Yaskawa INFORM job: DEMO_ROOF_SIDE_0625_3PAINT_58.JBI

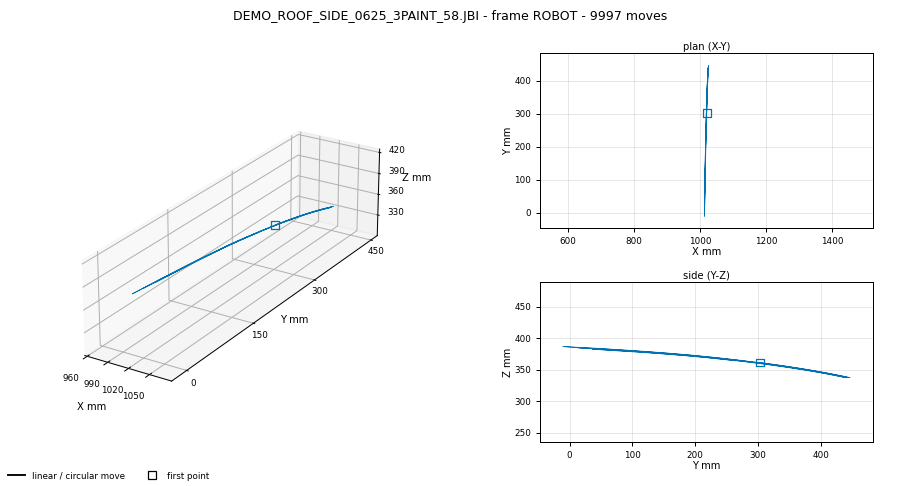
[picture p0: tool path of DEMO_ROOF_SIDE_0625_3PAINT_58.JBI in frame ROBOT, 9997 of 9997 moves have a stored position in this frame; points joined in program order, loops and branches not executed]
/JOB
//NAME DEMO_ROOF_SIDE_0625_3PAINT58
//POS
///NPOS 9997,0,0,0,0,0
///TOOL 0
///USER 0
///POSTYPE ROBOT
///RECTAN
///RCONF 1,0,0,0,0,0,0,0,0,0,0,0,0,0,0,0,0,0,0,0,0,0,0,0
C00000=1019.458,302.892,361.621,170.193,50.128,159.718
C00001=1019.464,303.141,361.589,170.199,50.124,159.718
C00002=1019.471,303.388,361.557,170.204,50.121,159.718
C00003=1019.478,303.636,361.524,170.209,50.117,159.718
C00004=1019.484,303.884,361.492,170.215,50.113,159.718
C00005=1019.491,304.131,361.460,170.220,50.110,159.718
C00006=1019.498,304.379,361.427,170.227,50.106,159.719
C00007=1019.504,304.627,361.396,170.232,50.103,159.719
C00008=1019.511,304.875,361.363,170.237,50.099,159.719
C00009=1019.517,305.122,361.330,170.243,50.095,159.719
C00010=1019.524,305.370,361.299,170.248,50.092,159.719
C00011=1019.530,305.618,361.266,170.255,50.088,159.719
C00012=1019.538,305.866,361.233,170.260,50.085,159.719
C00013=1019.544,306.113,361.201,170.265,50.082,159.719
C00014=1019.550,306.362,361.169,170.271,50.077,159.719
C00015=1019.557,306.609,361.136,170.276,50.074,159.719
C00016=1019.564,306.857,361.103,170.283,50.070,159.720
C00017=1019.570,307.101,361.071,170.288,50.067,159.720
C00018=1019.576,307.344,361.040,170.293,50.064,159.720
C00019=1019.583,307.587,361.008,170.299,50.060,159.720
C00020=1019.590,307.830,360.975,170.305,50.057,159.720
C00021=1019.596,308.074,360.944,170.310,50.053,159.720
C00022=1019.604,308.318,360.911,170.316,50.050,159.720
C00023=1019.610,308.562,360.879,170.322,50.046,159.720
C00024=1019.617,308.805,360.848,170.327,50.043,159.721
C00025=1019.624,309.052,360.815,170.333,50.039,159.721
C00026=1019.630,309.300,360.783,170.338,50.036,159.721
C00027=1019.637,309.548,360.750,170.345,50.033,159.721
C00028=1019.644,309.796,360.717,170.350,50.029,159.721
C00029=1019.650,310.043,360.685,170.356,50.026,159.721
C00030=1019.658,310.291,360.651,170.362,50.023,159.722
C00031=1019.663,310.539,360.618,170.367,50.020,159.722
C00032=1019.669,310.786,360.585,170.373,50.016,159.722
C00033=1019.677,311.034,360.551,170.379,50.013,159.722
C00034=1019.683,311.282,360.518,170.384,50.010,159.722
C00035=1019.689,311.529,360.485,170.391,50.007,159.723
C00036=1019.696,311.777,360.451,170.396,50.004,159.723
C00037=1019.702,312.025,360.418,170.402,50.000,159.723
C00038=1019.709,312.272,360.385,170.408,49.997,159.723
C00039=1019.715,312.520,360.352,170.414,49.994,159.723
C00040=1019.721,312.767,360.318,170.419,49.991,159.724
C00041=1019.728,313.015,360.285,170.425,49.988,159.724
C00042=1019.735,313.263,360.251,170.431,49.984,159.724
C00043=1019.741,313.510,360.218,170.437,49.981,159.724
C00044=1019.748,313.758,360.184,170.443,49.978,159.724
C00045=1019.754,314.006,360.151,170.448,49.976,159.725
C00046=1019.761,314.254,360.117,170.455,49.972,159.725
C00047=1019.768,314.500,360.084,170.460,49.969,159.725
C00048=1019.775,314.749,360.051,170.466,49.967,159.726
C00049=1019.780,314.996,360.017,170.472,49.963,159.726
C00050=1019.788,315.244,359.983,170.478,49.960,159.726
C00051=1019.794,315.491,359.950,170.484,49.957,159.726
C00052=1019.801,315.739,359.916,170.490,49.954,159.727
C00053=1019.807,315.986,359.882,170.495,49.951,159.727
C00054=1019.814,316.235,359.849,170.502,49.948,159.727
C00055=1019.820,316.482,359.816,170.507,49.945,159.727
C00056=1019.828,316.729,359.782,170.514,49.941,159.728
C00057=1019.834,316.977,359.748,170.519,49.939,159.728
C00058=1019.840,317.225,359.715,170.526,49.936,159.728
C00059=1019.848,317.472,359.681,170.532,49.933,159.729
C00060=1019.854,317.719,359.648,170.537,49.930,159.729
C00061=1019.861,317.967,359.613,170.544,49.927,159.729
C00062=1019.868,318.215,359.579,170.549,49.924,159.729
C00063=1019.874,318.462,359.546,170.556,49.921,159.730
C00064=1019.881,318.710,359.513,170.561,49.918,159.730
C00065=1019.888,318.958,359.478,170.568,49.915,159.730
C00066=1019.894,319.205,359.445,170.574,49.912,159.731
C00067=1019.902,319.453,359.411,170.580,49.909,159.731
C00068=1019.909,319.701,359.377,170.586,49.907,159.731
C00069=1019.915,319.949,359.343,170.591,49.903,159.731
C00070=1019.922,320.196,359.309,170.598,49.900,159.732
C00071=1019.929,320.443,359.275,170.603,49.898,159.732
C00072=1019.936,320.691,359.241,170.610,49.895,159.732
C00073=1019.943,320.939,359.207,170.616,49.892,159.733
C00074=1019.950,321.187,359.173,170.622,49.889,159.733
C00075=1019.957,321.434,359.140,170.628,49.886,159.733
C00076=1019.963,321.682,359.106,170.635,49.883,159.734
C00077=1019.971,321.928,359.072,170.640,49.881,159.734
C00078=1019.978,322.174,359.038,170.647,49.878,159.734
C00079=1019.984,322.420,359.004,170.653,49.875,159.735
C00080=1019.991,322.666,358.970,170.659,49.872,159.735
C00081=1019.998,322.912,358.936,170.665,49.869,159.735
C00082=1020.005,323.158,358.902,170.672,49.866,159.736
C00083=1020.012,323.404,358.868,170.677,49.864,159.736
C00084=1020.019,323.650,358.835,170.684,49.861,159.736
C00085=1020.026,323.898,358.800,170.690,49.858,159.737
C00086=1020.033,324.146,358.766,170.696,49.855,159.737
C00087=1020.040,324.393,358.732,170.702,49.853,159.737
C00088=1020.047,324.641,358.697,170.709,49.850,159.738
C00089=1020.054,324.888,358.664,170.715,49.848,159.738
C00090=1020.062,325.135,358.629,170.721,49.845,159.739
C00091=1020.069,325.383,358.595,170.727,49.842,159.739
C00092=1020.075,325.631,358.561,170.734,49.839,159.739
C00093=1020.083,325.878,358.526,170.739,49.836,159.740
C00094=1020.090,326.126,358.492,170.746,49.834,159.740
C00095=1020.097,326.373,358.458,170.753,49.831,159.741
C00096=1020.104,326.621,358.424,170.758,49.828,159.741
C00097=1020.111,326.868,358.388,170.766,49.826,159.741
C00098=1020.118,327.115,358.354,170.771,49.823,159.742
C00099=1020.125,327.363,358.319,170.778,49.821,159.742
C00100=1020.131,327.611,358.284,170.784,49.818,159.743
C00101=1020.139,327.858,358.250,170.791,49.815,159.743
C00102=1020.145,328.106,358.215,170.797,49.813,159.744
C00103=1020.152,328.353,358.180,170.803,49.810,159.744
C00104=1020.159,328.600,358.145,170.809,49.808,159.744
C00105=1020.167,328.848,358.110,170.816,49.806,159.745
C00106=1020.174,329.095,358.075,170.822,49.803,159.745
C00107=1020.181,329.343,358.040,170.829,49.801,159.746
C00108=1020.187,329.591,358.005,170.835,49.798,159.746
C00109=1020.195,329.838,357.971,170.842,49.796,159.747
C00110=1020.201,330.085,357.936,170.848,49.794,159.747
C00111=1020.208,330.333,357.901,170.854,49.791,159.748
C00112=1020.216,330.580,357.866,170.860,49.789,159.748
C00113=1020.223,330.828,357.831,170.867,49.786,159.748
C00114=1020.230,331.075,357.795,170.873,49.784,159.749
C00115=1020.237,331.322,357.760,170.880,49.782,159.750
C00116=1020.244,331.569,357.726,170.887,49.779,159.750
C00117=1020.251,331.818,357.690,170.893,49.777,159.750
C00118=1020.258,332.065,357.655,170.900,49.774,159.751
C00119=1020.265,332.312,357.620,170.906,49.772,159.751
C00120=1020.273,332.560,357.585,170.913,49.770,159.752
C00121=1020.280,332.807,357.550,170.919,49.767,159.752
C00122=1020.287,333.054,357.514,170.925,49.765,159.753
C00123=1020.294,333.301,357.479,170.932,49.763,159.753
C00124=1020.301,333.550,357.443,170.939,49.761,159.754
C00125=1020.308,333.796,357.408,170.946,49.758,159.755
C00126=1020.315,334.044,357.373,170.952,49.756,159.755
C00127=1020.322,334.292,357.337,170.959,49.754,159.756
C00128=1020.329,334.538,357.301,170.965,49.752,159.756
C00129=1020.336,334.786,357.266,170.972,49.750,159.757
C00130=1020.343,335.034,357.231,170.979,49.747,159.757
C00131=1020.351,335.281,357.195,170.985,49.745,159.758
C00132=1020.357,335.528,357.160,170.992,49.743,159.758
C00133=1020.365,335.775,357.123,170.998,49.741,159.759
C00134=1020.372,336.023,357.088,171.005,49.739,159.759
C00135=1020.379,336.270,357.052,171.012,49.736,159.760
C00136=1020.386,336.518,357.017,171.018,49.734,159.760
C00137=1020.393,336.762,356.982,171.025,49.733,159.761
C00138=1020.401,337.005,356.946,171.031,49.731,159.762
C00139=1020.408,337.250,356.911,171.038,49.728,159.762
C00140=1020.415,337.493,356.875,171.044,49.726,159.763
C00141=1020.422,337.737,356.841,171.051,49.724,159.763
C00142=1020.429,337.981,356.806,171.058,49.723,159.764
C00143=1020.436,338.225,356.770,171.065,49.720,159.765
C00144=1020.444,338.469,356.735,171.072,49.718,159.765
C00145=1020.451,338.716,356.699,171.078,49.716,159.766
C00146=1020.459,338.963,356.663,171.085,49.714,159.766
C00147=1020.466,339.211,356.628,171.092,49.712,159.767
C00148=1020.473,339.458,356.592,171.098,49.710,159.768
C00149=1020.480,339.705,356.555,171.106,49.708,159.768
C00150=1020.487,339.953,356.519,171.113,49.706,159.769
C00151=1020.495,340.200,356.483,171.119,49.704,159.770
C00152=1020.502,340.447,356.447,171.126,49.702,159.770
C00153=1020.509,340.695,356.410,171.132,49.701,159.771
C00154=1020.516,340.941,356.374,171.139,49.698,159.771
C00155=1020.524,341.189,356.338,171.147,49.697,159.772
C00156=1020.531,341.436,356.302,171.153,49.695,159.773
C00157=1020.538,341.683,356.265,171.160,49.693,159.773
C00158=1020.545,341.931,356.229,171.167,49.691,159.774
C00159=1020.553,342.178,356.193,171.175,49.689,159.775
C00160=1020.561,342.426,356.157,171.181,49.687,159.775
C00161=1020.567,342.673,356.120,171.188,49.685,159.776
C00162=1020.575,342.919,356.083,171.195,49.684,159.777
C00163=1020.583,343.167,356.047,171.201,49.682,159.777
C00164=1020.590,343.415,356.010,171.209,49.680,159.778
C00165=1020.597,343.661,355.974,171.216,49.678,159.779
C00166=1020.605,343.908,355.937,171.223,49.677,159.780
C00167=1020.612,344.156,355.901,171.230,49.674,159.780
C00168=1020.619,344.403,355.864,171.237,49.673,159.781
C00169=1020.627,344.650,355.827,171.244,49.671,159.782
C00170=1020.634,344.897,355.791,171.251,49.670,159.782
C00171=1020.641,345.145,355.755,171.258,49.668,159.783
C00172=1020.649,345.392,355.718,171.265,49.666,159.784
C00173=1020.656,345.639,355.681,171.273,49.664,159.784
C00174=1020.664,345.886,355.644,171.279,49.662,159.785
C00175=1020.672,346.134,355.608,171.286,49.661,159.786
C00176=1020.679,346.381,355.570,171.294,49.659,159.787
C00177=1020.687,346.628,355.534,171.301,49.657,159.787
C00178=1020.695,346.875,355.497,171.308,49.656,159.788
C00179=1020.701,347.122,355.461,171.315,49.654,159.789
C00180=1020.709,347.369,355.424,171.322,49.653,159.790
C00181=1020.716,347.617,355.387,171.330,49.651,159.790
C00182=1020.724,347.863,355.350,171.337,49.649,159.791
C00183=1020.731,348.111,355.313,171.344,49.648,159.792
C00184=1020.739,348.357,355.276,171.351,49.646,159.793
C00185=1020.746,348.605,355.239,171.358,49.644,159.793
C00186=1020.754,348.852,355.201,171.366,49.643,159.794
C00187=1020.762,349.099,355.164,171.374,49.642,159.795
C00188=1020.769,349.346,355.127,171.380,49.640,159.796
C00189=1020.777,349.593,355.090,171.387,49.638,159.797
C00190=1020.784,349.840,355.052,171.395,49.637,159.797
C00191=1020.792,350.088,355.014,171.402,49.636,159.798
C00192=1020.800,350.335,354.978,171.410,49.634,159.799
C00193=1020.807,350.582,354.940,171.416,49.633,159.800
C00194=1020.815,350.829,354.903,171.424,49.631,159.801
C00195=1020.822,351.076,354.866,171.431,49.630,159.802
C00196=1020.830,351.323,354.828,171.439,49.628,159.802
C00197=1020.837,351.560,354.793,171.447,49.627,159.803
C00198=1020.844,351.797,354.757,171.453,49.626,159.804
C00199=1020.851,352.033,354.721,171.460,49.624,159.805
C00200=1020.859,352.270,354.685,171.467,49.623,159.806
C00201=1020.866,352.506,354.649,171.474,49.621,159.806
C00202=1020.874,352.743,354.614,171.482,49.620,159.807
C00203=1020.881,352.980,354.577,171.489,49.619,159.808
C00204=1020.888,353.217,354.541,171.496,49.618,159.809
C00205=1020.897,353.463,354.503,171.504,49.616,159.810
C00206=1020.904,353.711,354.466,171.511,49.615,159.811
C00207=1020.912,353.958,354.428,171.519,49.613,159.812
C00208=1020.920,354.204,354.391,171.526,49.613,159.813
C00209=1020.928,354.452,354.353,171.533,49.611,159.813
C00210=1020.935,354.699,354.315,171.541,49.610,159.814
C00211=1020.943,354.945,354.277,171.549,49.609,159.815
C00212=1020.950,355.193,354.239,171.556,49.608,159.816
C00213=1020.959,355.439,354.201,171.564,49.606,159.817
C00214=1020.966,355.687,354.164,171.571,49.605,159.818
C00215=1020.974,355.934,354.125,171.579,49.604,159.819
C00216=1020.982,356.180,354.087,171.587,49.603,159.820
C00217=1020.990,356.440,354.048,171.595,49.601,159.821
C00218=1020.998,356.698,354.008,171.602,49.600,159.822
C00219=1021.006,356.956,353.969,171.611,49.599,159.823
C00220=1021.014,357.214,353.928,171.619,49.598,159.824
C00221=1021.023,357.461,353.890,171.626,49.596,159.825
C00222=1021.031,357.708,353.852,171.634,49.595,159.826
C00223=1021.038,357.955,353.814,171.642,49.594,159.827
C00224=1021.046,358.202,353.776,171.650,49.593,159.827
C00225=1021.054,358.449,353.737,171.657,49.592,159.828
C00226=1021.062,358.696,353.699,171.665,49.591,159.829
C00227=1021.069,358.942,353.660,171.673,49.590,159.830
C00228=1021.078,359.190,353.622,171.681,49.589,159.832
C00229=1021.086,359.436,353.584,171.689,49.588,159.833
C00230=1021.094,359.683,353.546,171.697,49.587,159.833
C00231=1021.102,359.930,353.507,171.704,49.586,159.834
C00232=1021.109,360.177,353.468,171.712,49.585,159.835
C00233=1021.117,360.424,353.430,171.720,49.584,159.836
C00234=1021.125,360.671,353.391,171.728,49.583,159.838
C00235=1021.133,360.918,353.353,171.736,49.582,159.839
C00236=1021.141,361.165,353.314,171.743,49.581,159.839
C00237=1021.149,361.411,353.275,171.752,49.580,159.841
C00238=1021.157,361.658,353.236,171.760,49.579,159.842
C00239=1021.164,361.906,353.197,171.768,49.578,159.843
C00240=1021.172,362.152,353.158,171.776,49.577,159.844
C00241=1021.180,362.399,353.120,171.784,49.576,159.845
C00242=1021.189,362.646,353.081,171.792,49.576,159.846
C00243=1021.196,362.892,353.042,171.800,49.575,159.847
C00244=1021.205,363.139,353.004,171.808,49.574,159.848
C00245=1021.213,363.386,352.964,171.816,49.573,159.849
C00246=1021.220,363.634,352.925,171.824,49.573,159.850
C00247=1021.229,363.881,352.886,171.833,49.571,159.851
C00248=1021.236,364.127,352.847,171.841,49.571,159.852
C00249=1021.245,364.373,352.808,171.848,49.570,159.853
C00250=1021.253,364.620,352.770,171.857,49.569,159.855
C00251=1021.261,364.867,352.730,171.865,49.569,159.856
C00252=1021.270,365.114,352.692,171.872,49.567,159.857
C00253=1021.277,365.361,352.652,171.882,49.567,159.858
C00254=1021.286,365.608,352.612,171.890,49.566,159.859
C00255=1021.293,365.854,352.574,171.897,49.565,159.860
C00256=1021.302,366.101,352.535,171.906,49.565,159.861
C00257=1021.310,366.347,352.495,171.914,49.564,159.862
C00258=1021.318,366.593,352.456,171.923,49.563,159.864
C00259=1021.327,366.838,352.417,171.931,49.563,159.865
C00260=1021.335,367.084,352.378,171.939,49.562,159.866
C00261=1021.343,367.331,352.339,171.947,49.561,159.867
C00262=1021.352,367.576,352.299,171.956,49.560,159.868
C00263=1021.359,367.822,352.261,171.964,49.560,159.869
C00264=1021.368,368.068,352.221,171.972,49.559,159.871
C00265=1021.377,368.314,352.181,171.980,49.559,159.872
C00266=1021.385,368.561,352.142,171.989,49.558,159.873
C00267=1021.393,368.808,352.102,171.997,49.557,159.874
C00268=1021.401,369.055,352.063,172.006,49.557,159.875
C00269=1021.409,369.301,352.023,172.014,49.556,159.877
C00270=1021.418,369.547,351.983,172.023,49.556,159.878
C00271=1021.425,369.794,351.943,172.031,49.556,159.879
C00272=1021.434,370.041,351.903,172.039,49.555,159.880
C00273=1021.442,370.288,351.863,172.049,49.554,159.882
C00274=1021.451,370.535,351.823,172.057,49.554,159.883
C00275=1021.459,370.781,351.783,172.065,49.554,159.884
C00276=1021.467,371.028,351.744,172.074,49.553,159.885
C00277=1021.475,371.274,351.703,172.082,49.553,159.887
C00278=1021.484,371.521,351.664,172.091,49.553,159.888
C00279=1021.492,371.768,351.623,172.100,49.552,159.889
C00280=1021.501,372.014,351.584,172.108,49.551,159.890
C00281=1021.509,372.261,351.543,172.117,49.551,159.892
C00282=1021.518,372.508,351.503,172.126,49.551,159.893
C00283=1021.526,372.754,351.463,172.134,49.551,159.894
C00284=1021.535,373.000,351.423,172.143,49.550,159.896
C00285=1021.543,373.248,351.382,172.152,49.550,159.897
C00286=1021.552,373.494,351.342,172.161,49.549,159.898
C00287=1021.560,373.740,351.302,172.169,49.549,159.900
C00288=1021.569,373.987,351.262,172.178,49.549,159.901
C00289=1021.577,374.234,351.221,172.187,49.548,159.902
C00290=1021.586,374.480,351.181,172.196,49.549,159.904
C00291=1021.594,374.727,351.140,172.205,49.548,159.905
C00292=1021.603,374.973,351.100,172.213,49.548,159.906
C00293=1021.611,375.220,351.060,172.223,49.548,159.908
C00294=1021.620,375.466,351.020,172.231,49.547,159.909
C00295=1021.629,375.713,350.979,172.240,49.547,159.910
C00296=1021.637,375.959,350.939,172.249,49.547,159.912
C00297=1021.646,376.206,350.898,172.258,49.547,159.913
C00298=1021.655,376.453,350.857,172.268,49.546,159.915
C00299=1021.664,376.699,350.816,172.276,49.546,159.916
C00300=1021.672,376.946,350.775,172.286,49.546,159.917
C00301=1021.680,377.192,350.734,172.294,49.546,159.919
C00302=1021.689,377.439,350.693,172.304,49.546,159.920
C00303=1021.697,377.684,350.652,172.312,49.546,159.922
C00304=1021.707,377.931,350.612,172.322,49.546,159.923
C00305=1021.715,378.177,350.571,172.330,49.546,159.924
C00306=1021.724,378.424,350.529,172.340,49.546,159.926
C00307=1021.732,378.671,350.488,172.349,49.545,159.927
C00308=1021.741,378.916,350.447,172.358,49.545,159.929
C00309=1021.749,379.163,350.406,172.367,49.545,159.930
C00310=1021.759,379.409,350.365,172.376,49.546,159.932
C00311=1021.768,379.656,350.324,172.385,49.546,159.933
C00312=1021.776,379.902,350.282,172.395,49.545,159.935
C00313=1021.785,380.149,350.241,172.404,49.546,159.936
C00314=1021.793,380.395,350.200,172.413,49.546,159.938
C00315=1021.802,380.642,350.159,172.423,49.546,159.939
C00316=1021.811,380.888,350.118,172.432,49.546,159.941
C00317=1021.821,381.155,350.072,172.442,49.546,159.942
C00318=1021.831,381.422,350.028,172.452,49.546,159.944
C00319=1021.840,381.689,349.983,172.463,49.546,159.946
C00320=1021.849,381.956,349.938,172.473,49.546,159.947
C00321=1021.858,382.202,349.897,172.482,49.546,159.949
C00322=1021.867,382.449,349.855,172.492,49.546,159.950
C00323=1021.877,382.695,349.814,172.501,49.547,159.952
C00324=1021.886,382.941,349.772,172.510,49.547,159.953
C00325=1021.895,383.188,349.730,172.520,49.547,159.955
C00326=1021.904,383.434,349.689,172.530,49.547,159.957
C00327=1021.913,383.680,349.647,172.540,49.547,159.958
C00328=1021.921,383.927,349.605,172.548,49.548,159.960
C00329=1021.931,384.173,349.564,172.558,49.548,159.961
C00330=1021.940,384.419,349.522,172.568,49.548,159.963
C00331=1021.949,384.665,349.481,172.578,49.548,159.965
C00332=1021.959,384.912,349.439,172.587,49.548,159.966
C00333=1021.968,385.158,349.396,172.597,49.549,159.968
C00334=1021.977,385.405,349.354,172.607,49.549,159.970
C00335=1021.986,385.651,349.313,172.617,49.549,159.971
C00336=1021.995,385.897,349.270,172.626,49.550,159.973
C00337=1022.004,386.143,349.229,172.636,49.550,159.974
C00338=1022.013,386.390,349.186,172.646,49.551,159.976
C00339=1022.023,386.636,349.144,172.655,49.551,159.978
C00340=1022.032,386.882,349.102,172.665,49.551,159.979
C00341=1022.041,387.128,349.060,172.675,49.552,159.981
C00342=1022.050,387.374,349.017,172.685,49.552,159.983
C00343=1022.060,387.621,348.975,172.695,49.552,159.984
C00344=1022.069,387.867,348.933,172.705,49.553,159.986
C00345=1022.077,388.113,348.890,172.715,49.553,159.988
C00346=1022.087,388.360,348.848,172.725,49.554,159.990
C00347=1022.096,388.605,348.805,172.735,49.555,159.991
C00348=1022.105,388.851,348.763,172.745,49.555,159.993
C00349=1022.115,389.098,348.720,172.755,49.555,159.995
C00350=1022.124,389.344,348.677,172.765,49.556,159.997
C00351=1022.133,389.589,348.635,172.775,49.557,159.998
C00352=1022.143,389.836,348.592,172.785,49.557,160.000
C00353=1022.152,390.082,348.549,172.796,49.557,160.002
C00354=1022.161,390.328,348.506,172.806,49.558,160.004
C00355=1022.170,390.574,348.464,172.816,49.559,160.005
C00356=1022.180,390.820,348.421,172.826,49.559,160.007
C00357=1022.189,391.066,348.378,172.836,49.560,160.009
C00358=1022.199,391.312,348.334,172.846,49.561,160.011
C00359=1022.208,391.558,348.292,172.856,49.561,160.013
C00360=1022.218,391.805,348.249,172.868,49.562,160.015
C00361=1022.227,392.050,348.207,172.878,49.563,160.017
C00362=1022.237,392.296,348.163,172.888,49.563,160.018
C00363=1022.246,392.542,348.120,172.898,49.564,160.020
C00364=1022.256,392.789,348.077,172.908,49.565,160.022
C00365=1022.265,393.035,348.033,172.919,49.565,160.024
C00366=1022.274,393.280,347.991,172.930,49.566,160.026
C00367=1022.284,393.526,347.947,172.940,49.567,160.028
C00368=1022.294,393.772,347.903,172.950,49.568,160.030
C00369=1022.303,394.018,347.861,172.961,49.569,160.031
C00370=1022.312,394.264,347.817,172.972,49.570,160.033
C00371=1022.323,394.510,347.773,172.982,49.570,160.035
C00372=1022.332,394.757,347.730,172.993,49.572,160.037
C00373=1022.341,395.002,347.687,173.004,49.572,160.039
C00374=1022.351,395.248,347.643,173.014,49.573,160.041
C00375=1022.361,395.494,347.599,173.025,49.574,160.043
C00376=1022.371,395.740,347.555,173.036,49.575,160.045
C00377=1022.382,396.044,347.501,173.048,49.576,160.047
C00378=1022.395,396.348,347.447,173.062,49.577,160.050
C00379=1022.407,396.652,347.393,173.075,49.578,160.052
C00380=1022.419,396.956,347.339,173.089,49.579,160.055
C00381=1022.429,397.203,347.295,173.100,49.581,160.057
C00382=1022.439,397.448,347.252,173.111,49.581,160.059
C00383=1022.448,397.694,347.207,173.122,49.583,160.061
C00384=1022.459,397.940,347.163,173.133,49.583,160.063
C00385=1022.468,398.186,347.119,173.143,49.585,160.065
C00386=1022.478,398.432,347.076,173.155,49.586,160.067
C00387=1022.488,398.677,347.031,173.165,49.587,160.069
C00388=1022.497,398.923,346.987,173.177,49.588,160.071
C00389=1022.508,399.168,346.943,173.188,49.589,160.073
C00390=1022.517,399.415,346.898,173.199,49.590,160.075
C00391=1022.527,399.660,346.854,173.209,49.591,160.077
C00392=1022.537,399.906,346.810,173.221,49.592,160.079
C00393=1022.547,400.152,346.765,173.233,49.593,160.082
C00394=1022.557,400.398,346.720,173.243,49.595,160.084
C00395=1022.567,400.644,346.677,173.255,49.596,160.086
C00396=1022.577,400.889,346.632,173.266,49.597,160.088
C00397=1022.587,401.135,346.587,173.277,49.598,160.090
C00398=1022.597,401.381,346.542,173.289,49.600,160.092
C00399=1022.607,401.626,346.498,173.301,49.601,160.095
C00400=1022.617,401.871,346.453,173.311,49.602,160.097
C00401=1022.627,402.118,346.408,173.323,49.603,160.099
C00402=1022.637,402.363,346.363,173.334,49.604,160.101
C00403=1022.647,402.609,346.318,173.346,49.606,160.103
C00404=1022.657,402.855,346.273,173.357,49.608,160.106
C00405=1022.668,403.100,346.228,173.369,49.609,160.108
C00406=1022.677,403.346,346.184,173.380,49.610,160.110
C00407=1022.688,403.592,346.138,173.392,49.611,160.112
C00408=1022.697,403.837,346.094,173.404,49.613,160.115
C00409=1022.708,404.083,346.048,173.415,49.614,160.117
C00410=1022.718,404.328,346.003,173.427,49.616,160.119
C00411=1022.728,404.575,345.958,173.439,49.618,160.121
C00412=1022.739,404.819,345.913,173.450,49.619,160.124
C00413=1022.749,405.065,345.868,173.462,49.620,160.126
C00414=1022.760,405.311,345.822,173.474,49.622,160.128
C00415=1022.769,405.557,345.777,173.486,49.623,160.130
C00416=1022.780,405.802,345.731,173.498,49.625,160.133
C00417=1022.790,406.048,345.686,173.510,49.626,160.135
C00418=1022.800,406.293,345.640,173.522,49.628,160.138
C00419=1022.812,406.539,345.595,173.534,49.629,160.140
C00420=1022.822,406.785,345.550,173.546,49.631,160.142
C00421=1022.833,407.030,345.504,173.558,49.633,160.145
C00422=1022.843,407.276,345.458,173.570,49.634,160.147
C00423=1022.853,407.521,345.412,173.582,49.636,160.150
C00424=1022.864,407.767,345.367,173.594,49.637,160.152
C00425=1022.874,408.013,345.321,173.607,49.639,160.154
C00426=1022.886,408.258,345.276,173.619,49.640,160.157
C00427=1022.896,408.504,345.230,173.631,49.642,160.159
C00428=1022.907,408.749,345.184,173.643,49.643,160.161
C00429=1022.918,408.995,345.138,173.655,49.646,160.164
C00430=1022.928,409.240,345.092,173.667,49.647,160.166
C00431=1022.939,409.486,345.046,173.680,49.648,160.169
C00432=1022.950,409.731,345.000,173.692,49.651,160.171
C00433=1022.960,409.976,344.954,173.704,49.652,160.174
C00434=1022.970,410.222,344.907,173.717,49.654,160.176
C00435=1022.981,410.467,344.861,173.729,49.655,160.179
C00436=1022.992,410.713,344.815,173.742,49.658,160.181
C00437=1023.007,411.039,344.753,173.758,49.661,160.185
C00438=1023.021,411.366,344.691,173.775,49.662,160.188
C00439=1023.035,411.692,344.629,173.792,49.665,160.192
C00440=1023.049,412.019,344.568,173.809,49.668,160.195
C00441=1023.060,412.264,344.521,173.821,49.669,160.198
C00442=1023.072,412.510,344.474,173.835,49.671,160.200
C00443=1023.082,412.755,344.427,173.847,49.673,160.203
C00444=1023.093,413.000,344.380,173.860,49.675,160.206
C00445=1023.104,413.246,344.334,173.873,49.677,160.208
C00446=1023.115,413.491,344.287,173.886,49.679,160.211
C00447=1023.126,413.736,344.241,173.899,49.682,160.214
C00448=1023.138,413.982,344.194,173.912,49.683,160.216
C00449=1023.148,414.227,344.146,173.925,49.686,160.219
C00450=1023.159,414.473,344.099,173.938,49.687,160.222
C00451=1023.170,414.718,344.053,173.951,49.689,160.224
C00452=1023.182,414.963,344.005,173.964,49.692,160.227
C00453=1023.193,415.208,343.958,173.977,49.693,160.230
C00454=1023.204,415.454,343.911,173.991,49.696,160.233
C00455=1023.215,415.700,343.864,174.004,49.698,160.235
C00456=1023.227,415.944,343.816,174.017,49.700,160.238
C00457=1023.237,416.190,343.769,174.031,49.702,160.241
C00458=1023.249,416.435,343.721,174.044,49.704,160.244
C00459=1023.259,416.680,343.674,174.057,49.707,160.246
C00460=1023.271,416.925,343.626,174.070,49.709,160.249
C00461=1023.282,417.171,343.578,174.084,49.711,160.252
C00462=1023.293,417.416,343.531,174.098,49.713,160.255
C00463=1023.304,417.661,343.483,174.112,49.716,160.258
C00464=1023.316,417.906,343.435,174.125,49.718,160.261
C00465=1023.327,418.152,343.387,174.138,49.721,160.264
C00466=1023.339,418.397,343.339,174.152,49.723,160.266
C00467=1023.351,418.642,343.292,174.166,49.725,160.269
C00468=1023.361,418.886,343.244,174.179,49.727,160.272
C00469=1023.373,419.131,343.196,174.193,49.730,160.275
C00470=1023.384,419.377,343.148,174.207,49.732,160.278
C00471=1023.396,419.622,343.100,174.221,49.734,160.281
C00472=1023.407,419.867,343.052,174.235,49.737,160.284
C00473=1023.419,420.112,343.004,174.249,49.739,160.287
C00474=1023.431,420.358,342.955,174.263,49.741,160.290
C00475=1023.443,420.603,342.907,174.277,49.744,160.293
C00476=1023.455,420.848,342.859,174.291,49.746,160.296
C00477=1023.466,421.093,342.811,174.305,49.749,160.299
C00478=1023.478,421.338,342.763,174.319,49.751,160.302
C00479=1023.490,421.584,342.714,174.334,49.754,160.305
C00480=1023.502,421.828,342.665,174.348,49.756,160.308
C00481=1023.513,422.073,342.617,174.362,49.759,160.311
C00482=1023.524,422.318,342.568,174.376,49.762,160.314
C00483=1023.537,422.563,342.519,174.391,49.764,160.317
C00484=1023.549,422.808,342.470,174.405,49.767,160.320
C00485=1023.560,423.053,342.422,174.420,49.770,160.324
C00486=1023.572,423.299,342.373,174.435,49.772,160.327
C00487=1023.584,423.543,342.324,174.449,49.775,160.330
C00488=1023.595,423.788,342.275,174.464,49.777,160.333
C00489=1023.608,424.033,342.226,174.478,49.780,160.336
C00490=1023.619,424.278,342.177,174.493,49.782,160.339
C00491=1023.632,424.523,342.127,174.507,49.785,160.342
C00492=1023.644,424.767,342.079,174.523,49.788,160.346
C00493=1023.656,425.013,342.030,174.537,49.791,160.349
C00494=1023.668,425.258,341.980,174.552,49.793,160.352
C00495=1023.679,425.503,341.931,174.568,49.796,160.355
C00496=1023.692,425.747,341.882,174.582,49.799,160.359
C00497=1023.709,426.085,341.813,174.603,49.803,160.363
C00498=1023.725,426.423,341.744,174.624,49.807,160.368
C00499=1023.742,426.762,341.676,174.644,49.811,160.372
C00500=1023.758,427.099,341.608,174.665,49.815,160.377
C00501=1023.771,427.344,341.558,174.681,49.818,160.380
C00502=1023.783,427.589,341.508,174.696,49.821,160.384
C00503=1023.796,427.833,341.458,174.712,49.824,160.387
C00504=1023.808,428.078,341.408,174.727,49.827,160.391
C00505=1023.821,428.323,341.358,174.743,49.830,160.394
C00506=1023.833,428.568,341.308,174.758,49.833,160.397
C00507=1023.845,428.812,341.258,174.774,49.836,160.401
C00508=1023.857,429.057,341.208,174.789,49.839,160.404
C00509=1023.869,429.301,341.158,174.805,49.841,160.408
C00510=1023.882,429.546,341.107,174.821,49.845,160.411
C00511=1023.895,429.791,341.057,174.836,49.848,160.415
C00512=1023.908,430.036,341.007,174.852,49.851,160.418
C00513=1023.920,430.280,340.956,174.868,49.854,160.422
C00514=1023.933,430.525,340.906,174.883,49.858,160.425
C00515=1023.945,430.769,340.855,174.899,49.860,160.429
C00516=1023.958,431.014,340.805,174.916,49.864,160.433
C00517=1023.971,431.259,340.754,174.932,49.867,160.436
C00518=1023.983,431.503,340.704,174.948,49.870,160.440
C00519=1023.996,431.748,340.653,174.964,49.873,160.443
C00520=1024.009,431.991,340.603,174.980,49.876,160.447
C00521=1024.022,432.236,340.552,174.996,49.880,160.451
C00522=1024.035,432.481,340.501,175.013,49.883,160.454
C00523=1024.048,432.726,340.451,175.029,49.886,160.458
C00524=1024.061,432.970,340.399,175.046,49.889,160.462
C00525=1024.074,433.215,340.348,175.062,49.893,160.465
C00526=1024.087,433.459,340.297,175.079,49.896,160.469
C00527=1024.100,433.704,340.246,175.095,49.899,160.473
C00528=1024.112,433.948,340.195,175.112,49.903,160.477
C00529=1024.125,434.193,340.143,175.128,49.906,160.480
C00530=1024.138,434.437,340.091,175.145,49.910,160.484
C00531=1024.151,434.681,340.040,175.162,49.913,160.488
C00532=1024.165,434.926,339.989,175.178,49.917,160.492
C00533=1024.178,435.169,339.937,175.196,49.920,160.496
C00534=1024.191,435.414,339.885,175.213,49.923,160.499
C00535=1024.204,435.659,339.834,175.230,49.927,160.503
C00536=1024.218,435.903,339.782,175.247,49.930,160.507
C00537=1024.230,436.147,339.730,175.264,49.934,160.511
C00538=1024.244,436.391,339.678,175.281,49.938,160.515
C00539=1024.257,436.635,339.626,175.298,49.941,160.519
C00540=1024.271,436.880,339.574,175.315,49.945,160.523
C00541=1024.284,437.124,339.522,175.333,49.949,160.527
C00542=1024.298,437.368,339.471,175.350,49.952,160.531
C00543=1024.311,437.613,339.419,175.368,49.956,160.535
C00544=1024.324,437.857,339.366,175.386,49.959,160.539
C00545=1024.338,438.101,339.314,175.404,49.963,160.543
C00546=1024.351,438.345,339.262,175.421,49.967,160.547
C00547=1024.365,438.589,339.209,175.439,49.970,160.551
C00548=1024.378,438.833,339.157,175.456,49.974,160.555
C00549=1024.392,439.077,339.104,175.475,49.978,160.560
C00550=1024.406,439.322,339.052,175.493,49.982,160.564
C00551=1024.420,439.566,338.999,175.510,49.985,160.568
C00552=1024.433,439.810,338.946,175.529,49.989,160.572
C00553=1024.447,440.053,338.893,175.546,49.993,160.576
C00554=1024.461,440.298,338.840,175.565,49.997,160.581
C00555=1024.475,440.541,338.788,175.583,50.001,160.585
C00556=1024.488,440.785,338.735,175.602,50.004,160.589
C00557=1024.511,441.179,338.649,175.631,50.011,160.596
C00558=1024.533,441.573,338.564,175.660,50.017,160.603
C00559=1024.556,441.966,338.479,175.691,50.023,160.610
C00560=1024.580,442.360,338.392,175.721,50.030,160.617
C00561=1024.594,442.603,338.340,175.739,50.034,160.621
C00562=1024.609,442.846,338.288,175.759,50.038,160.625
C00563=1024.625,443.089,338.236,175.777,50.041,160.630
C00564=1024.641,443.334,338.185,175.797,50.044,160.634
C00565=1024.657,443.577,338.134,175.816,50.048,160.638
C00566=1024.673,443.820,338.083,175.835,50.052,160.643
C00567=1024.691,444.064,338.032,175.855,50.055,160.647
C00568=1024.709,444.309,337.982,175.873,50.059,160.651
C00569=1024.726,444.552,337.933,175.893,50.062,160.656
C00570=1024.746,444.796,337.884,175.912,50.065,160.660
C00571=1024.765,445.040,337.835,175.932,50.068,160.664
C00572=1024.784,445.285,337.786,175.952,50.072,160.669
C00573=1024.805,445.529,337.739,175.972,50.075,160.673
C00574=1024.824,445.773,337.691,175.991,50.078,160.677
C00575=1024.845,446.017,337.644,176.012,50.080,160.681
C00576=1024.867,446.262,337.597,176.032,50.083,160.686
C00577=1024.405,444.052,337.704,175.845,50.118,160.665
C00578=1024.388,443.808,337.754,175.826,50.114,160.660
C00579=1024.371,443.564,337.804,175.807,50.111,160.656
C00580=1024.355,443.320,337.855,175.788,50.108,160.652
C00581=1024.339,443.077,337.907,175.769,50.104,160.648
C00582=1024.318,442.749,337.976,175.743,50.099,160.642
C00583=1024.298,442.421,338.047,175.718,50.094,160.636
C00584=1024.279,442.095,338.118,175.693,50.090,160.630
C00585=1024.259,441.768,338.189,175.668,50.084,160.624
C00586=1024.247,441.550,338.236,175.651,50.080,160.620
C00587=1024.235,441.332,338.284,175.634,50.078,160.617
C00588=1024.222,441.115,338.331,175.618,50.074,160.613
C00589=1024.209,440.897,338.378,175.602,50.070,160.609
C00590=1024.196,440.653,338.431,175.583,50.067,160.605
C00591=1024.182,440.409,338.484,175.565,50.063,160.601
C00592=1024.168,440.165,338.537,175.547,50.059,160.596
C00593=1024.154,439.921,338.590,175.528,50.056,160.592
C00594=1024.140,439.677,338.642,175.511,50.052,160.588
C00595=1024.127,439.433,338.694,175.493,50.048,160.584
C00596=1024.113,439.188,338.748,175.474,50.045,160.580
C00597=1024.099,438.945,338.801,175.456,50.041,160.576
C00598=1024.086,438.701,338.852,175.438,50.038,160.572
C00599=1024.072,438.457,338.905,175.420,50.034,160.567
C00600=1024.059,438.212,338.958,175.403,50.030,160.563
C00601=1024.045,437.969,339.010,175.385,50.026,160.559
C00602=1024.032,437.724,339.062,175.368,50.023,160.555
C00603=1024.018,437.480,339.114,175.350,50.020,160.551
C00604=1024.005,437.236,339.166,175.332,50.016,160.547
C00605=1023.991,436.991,339.218,175.315,50.012,160.543
C00606=1023.978,436.747,339.270,175.297,50.009,160.539
C00607=1023.965,436.503,339.322,175.280,50.005,160.535
C00608=1023.951,436.258,339.374,175.263,50.002,160.531
C00609=1023.938,436.014,339.426,175.246,49.999,160.528
C00610=1023.925,435.770,339.477,175.229,49.995,160.524
C00611=1023.911,435.526,339.529,175.211,49.992,160.520
C00612=1023.898,435.281,339.580,175.194,49.988,160.516
C00613=1023.885,435.037,339.633,175.178,49.985,160.512
C00614=1023.872,434.793,339.684,175.161,49.981,160.508
C00615=1023.859,434.548,339.736,175.144,49.979,160.504
C00616=1023.846,434.303,339.787,175.126,49.975,160.501
C00617=1023.833,434.060,339.838,175.111,49.972,160.497
C00618=1023.820,433.815,339.890,175.093,49.968,160.493
C00619=1023.807,433.571,339.940,175.076,49.965,160.489
C00620=1023.794,433.326,339.992,175.060,49.962,160.486
C00621=1023.781,433.082,340.043,175.043,49.959,160.482
C00622=1023.768,432.837,340.094,175.028,49.955,160.478
C00623=1023.755,432.593,340.145,175.011,49.952,160.474
C00624=1023.742,432.348,340.196,174.995,49.949,160.471
C00625=1023.729,432.104,340.247,174.978,49.946,160.467
C00626=1023.717,431.858,340.298,174.962,49.943,160.463
C00627=1023.704,431.614,340.348,174.945,49.940,160.460
C00628=1023.691,431.370,340.399,174.929,49.937,160.456
C00629=1023.679,431.125,340.449,174.913,49.933,160.453
C00630=1023.665,430.881,340.500,174.897,49.930,160.449
C00631=1023.652,430.636,340.551,174.881,49.927,160.446
C00632=1023.640,430.392,340.601,174.865,49.924,160.442
C00633=1023.628,430.147,340.651,174.849,49.922,160.438
C00634=1023.615,429.903,340.702,174.833,49.919,160.435
C00635=1023.603,429.658,340.752,174.817,49.915,160.431
C00636=1023.591,429.413,340.802,174.802,49.912,160.428
C00637=1023.577,429.169,340.852,174.786,49.909,160.424
C00638=1023.565,428.924,340.902,174.771,49.907,160.421
C00639=1023.553,428.679,340.952,174.755,49.904,160.418
C00640=1023.540,428.435,341.002,174.739,49.901,160.414
C00641=1023.528,428.190,341.052,174.724,49.898,160.411
C00642=1023.516,427.945,341.102,174.708,49.895,160.407
C00643=1023.503,427.700,341.153,174.693,49.892,160.404
C00644=1023.491,427.455,341.203,174.677,49.889,160.401
C00645=1023.478,427.211,341.252,174.662,49.886,160.397
C00646=1023.461,426.871,341.321,174.641,49.883,160.393
C00647=1023.445,426.530,341.391,174.620,49.879,160.388
C00648=1023.429,426.190,341.459,174.599,49.875,160.383
C00649=1023.411,425.850,341.529,174.578,49.871,160.379
C00650=1023.400,425.605,341.578,174.562,49.868,160.375
C00651=1023.387,425.360,341.627,174.548,49.865,160.372
C00652=1023.375,425.115,341.676,174.532,49.862,160.369
C00653=1023.364,424.870,341.725,174.517,49.860,160.366
C00654=1023.351,424.625,341.774,174.503,49.857,160.363
C00655=1023.339,424.380,341.823,174.488,49.855,160.359
C00656=1023.327,424.135,341.873,174.474,49.852,160.356
C00657=1023.315,423.891,341.922,174.459,49.850,160.353
C00658=1023.303,423.646,341.971,174.444,49.847,160.350
C00659=1023.291,423.401,342.020,174.429,49.845,160.347
C00660=1023.279,423.155,342.068,174.414,49.842,160.343
C00661=1023.268,422.910,342.117,174.400,49.839,160.340
C00662=1023.256,422.666,342.166,174.386,49.837,160.337
C00663=1023.244,422.421,342.215,174.371,49.835,160.334
C00664=1023.232,422.176,342.264,174.357,49.832,160.331
C00665=1023.220,421.931,342.312,174.343,49.829,160.328
C00666=1023.209,421.686,342.361,174.328,49.827,160.325
C00667=1023.198,421.441,342.409,174.314,49.825,160.322
C00668=1023.185,421.195,342.458,174.300,49.822,160.319
C00669=1023.174,420.950,342.506,174.285,49.820,160.316
C00670=1023.162,420.705,342.554,174.271,49.818,160.313
C00671=1023.150,420.461,342.602,174.257,49.815,160.310
C00672=1023.139,420.215,342.651,174.243,49.813,160.307
C00673=1023.127,419.970,342.698,174.230,49.810,160.304
C00674=1023.116,419.725,342.747,174.215,49.808,160.301
C00675=1023.104,419.480,342.794,174.201,49.806,160.298
C00676=1023.093,419.235,342.843,174.187,49.804,160.295
C00677=1023.081,418.990,342.891,174.174,49.802,160.292
C00678=1023.069,418.745,342.939,174.160,49.799,160.289
C00679=1023.058,418.499,342.987,174.146,49.797,160.287
C00680=1023.046,418.254,343.034,174.132,49.795,160.284
C00681=1023.035,418.008,343.082,174.119,49.793,160.281
C00682=1023.023,417.763,343.130,174.105,49.790,160.278
C00683=1023.013,417.519,343.178,174.091,49.788,160.275
C00684=1023.001,417.274,343.226,174.077,49.786,160.272
C00685=1022.990,417.028,343.273,174.064,49.784,160.269
C00686=1022.979,416.783,343.321,174.050,49.782,160.266
C00687=1022.968,416.538,343.367,174.038,49.779,160.264
C00688=1022.956,416.292,343.416,174.024,49.777,160.261
C00689=1022.945,416.047,343.463,174.010,49.775,160.258
C00690=1022.934,415.802,343.511,173.997,49.773,160.255
C00691=1022.923,415.556,343.558,173.983,49.771,160.252
C00692=1022.912,415.312,343.605,173.971,49.769,160.250
C00693=1022.901,415.066,343.653,173.958,49.767,160.247
C00694=1022.889,414.820,343.700,173.944,49.765,160.244
C00695=1022.878,414.575,343.746,173.931,49.763,160.242
C00696=1022.867,414.330,343.793,173.918,49.761,160.239
C00697=1022.856,414.085,343.840,173.905,49.759,160.236
C00698=1022.845,413.839,343.887,173.892,49.757,160.234
C00699=1022.834,413.594,343.934,173.879,49.755,160.231
C00700=1022.823,413.349,343.981,173.866,49.754,160.228
C00701=1022.812,413.103,344.028,173.853,49.752,160.226
C00702=1022.801,412.858,344.074,173.840,49.750,160.223
C00703=1022.790,412.613,344.121,173.827,49.748,160.220
C00704=1022.779,412.367,344.168,173.814,49.746,160.218
C00705=1022.769,412.122,344.214,173.802,49.744,160.215
C00706=1022.754,411.793,344.277,173.785,49.742,160.212
C00707=1022.739,411.464,344.339,173.767,49.739,160.208
C00708=1022.725,411.135,344.401,173.751,49.737,160.205
C00709=1022.711,410.806,344.464,173.733,49.735,160.201
C00710=1022.700,410.561,344.510,173.721,49.733,160.199
C00711=1022.689,410.315,344.557,173.708,49.731,160.196
C00712=1022.678,410.070,344.603,173.696,49.730,160.194
C00713=1022.667,409.824,344.649,173.684,49.728,160.191
C00714=1022.657,409.579,344.695,173.671,49.726,160.189
C00715=1022.647,409.333,344.742,173.659,49.725,160.187
C00716=1022.636,409.088,344.788,173.646,49.723,160.184
C00717=1022.625,408.842,344.833,173.634,49.721,160.182
C00718=1022.614,408.597,344.879,173.621,49.720,160.179
C00719=1022.603,408.351,344.925,173.609,49.718,160.177
C00720=1022.593,408.105,344.971,173.597,49.717,160.174
C00721=1022.582,407.860,345.016,173.585,49.715,160.172
C00722=1022.572,407.615,345.062,173.572,49.714,160.170
C00723=1022.562,407.369,345.107,173.560,49.712,160.167
C00724=1022.550,407.124,345.153,173.548,49.711,160.165
C00725=1022.540,406.878,345.198,173.536,49.709,160.162
C00726=1022.529,406.632,345.244,173.524,49.707,160.160
C00727=1022.520,406.387,345.289,173.513,49.706,160.158
C00728=1022.509,406.141,345.335,173.501,49.705,160.155
C00729=1022.499,405.895,345.380,173.489,49.703,160.153
C00730=1022.488,405.649,345.426,173.477,49.702,160.151
C00731=1022.478,405.404,345.470,173.464,49.701,160.148
C00732=1022.467,405.159,345.516,173.452,49.699,160.146
C00733=1022.457,404.913,345.561,173.441,49.698,160.144
C00734=1022.447,404.667,345.607,173.430,49.696,160.142
C00735=1022.436,404.421,345.652,173.418,49.695,160.139
C00736=1022.427,404.176,345.697,173.406,49.694,160.137
C00737=1022.415,403.930,345.742,173.394,49.693,160.135
C00738=1022.405,403.685,345.787,173.382,49.691,160.132
C00739=1022.396,403.439,345.832,173.371,49.690,160.130
C00740=1022.385,403.193,345.877,173.359,49.688,160.128
C00741=1022.375,402.948,345.923,173.347,49.687,160.126
C00742=1022.365,402.702,345.968,173.336,49.686,160.124
C00743=1022.355,402.457,346.012,173.325,49.685,160.121
C00744=1022.345,402.211,346.057,173.313,49.683,160.119
C00745=1022.335,401.965,346.102,173.301,49.682,160.117
C00746=1022.325,401.720,346.147,173.290,49.681,160.115
C00747=1022.315,401.474,346.192,173.278,49.680,160.113
C00748=1022.305,401.227,346.236,173.268,49.679,160.110
C00749=1022.295,400.982,346.281,173.256,49.678,160.108
C00750=1022.285,400.737,346.325,173.244,49.677,160.106
C00751=1022.275,400.491,346.370,173.233,49.676,160.104
C00752=1022.265,400.245,346.414,173.222,49.674,160.102
C00753=1022.255,399.999,346.459,173.210,49.673,160.100
C00754=1022.245,399.754,346.504,173.199,49.673,160.098
C00755=1022.235,399.508,346.547,173.189,49.671,160.096
C00756=1022.225,399.262,346.592,173.177,49.670,160.093
C00757=1022.216,399.016,346.636,173.165,49.669,160.091
C00758=1022.205,398.771,346.680,173.155,49.668,160.089
C00759=1022.196,398.525,346.724,173.144,49.667,160.087
C00760=1022.187,398.279,346.769,173.133,49.666,160.085
C00761=1022.176,398.033,346.813,173.122,49.665,160.083
C00762=1022.167,397.787,346.857,173.111,49.664,160.081
C00763=1022.157,397.541,346.900,173.100,49.663,160.079
C00764=1022.147,397.295,346.945,173.088,49.662,160.077
C00765=1022.137,397.050,346.988,173.078,49.661,160.075
C00766=1022.124,396.743,347.043,173.064,49.660,160.073
C00767=1022.112,396.437,347.097,173.051,49.659,160.070
C00768=1022.101,396.131,347.152,173.037,49.658,160.068
C00769=1022.088,395.823,347.207,173.024,49.657,160.065
C00770=1022.079,395.578,347.250,173.013,49.657,160.063
C00771=1022.069,395.332,347.294,173.003,49.655,160.061
C00772=1022.059,395.086,347.337,172.991,49.655,160.059
C00773=1022.049,394.840,347.380,172.981,49.654,160.057
C00774=1022.040,394.594,347.424,172.970,49.654,160.055
C00775=1022.030,394.349,347.467,172.960,49.653,160.054
C00776=1022.021,394.103,347.511,172.949,49.652,160.052
C00777=1022.011,393.856,347.554,172.938,49.651,160.050
C00778=1022.002,393.611,347.598,172.928,49.650,160.048
C00779=1021.992,393.364,347.641,172.918,49.650,160.046
C00780=1021.982,393.118,347.684,172.906,49.649,160.044
C00781=1021.973,392.873,347.728,172.896,49.648,160.042
C00782=1021.964,392.627,347.771,172.886,49.648,160.040
C00783=1021.954,392.380,347.814,172.876,49.647,160.039
C00784=1021.945,392.135,347.857,172.865,49.647,160.037
C00785=1021.935,391.888,347.900,172.855,49.646,160.035
C00786=1021.926,391.642,347.943,172.845,49.645,160.033
C00787=1021.916,391.396,347.985,172.834,49.645,160.031
C00788=1021.907,391.149,348.029,172.824,49.645,160.029
C00789=1021.897,390.904,348.072,172.813,49.644,160.028
C00790=1021.888,390.658,348.114,172.803,49.643,160.026
C00791=1021.878,390.412,348.157,172.793,49.643,160.024
C00792=1021.870,390.166,348.200,172.783,49.642,160.022
C00793=1021.860,389.919,348.243,172.772,49.642,160.020
C00794=1021.851,389.674,348.285,172.762,49.641,160.019
C00795=1021.841,389.427,348.328,172.752,49.641,160.017
C00796=1021.832,389.181,348.371,172.742,49.640,160.015
C00797=1021.823,388.935,348.414,172.732,49.640,160.014
C00798=1021.813,388.689,348.457,172.722,49.639,160.012
C00799=1021.804,388.443,348.498,172.712,49.639,160.010
C00800=1021.795,388.197,348.541,172.702,49.639,160.008
C00801=1021.786,387.950,348.584,172.692,49.639,160.007
C00802=1021.777,387.704,348.626,172.681,49.638,160.005
C00803=1021.768,387.458,348.668,172.671,49.637,160.003
C00804=1021.759,387.212,348.711,172.662,49.637,160.001
C00805=1021.749,386.965,348.753,172.652,49.637,160.000
C00806=1021.740,386.720,348.795,172.642,49.636,159.998
C00807=1021.731,386.473,348.837,172.632,49.636,159.996
C00808=1021.722,386.227,348.879,172.622,49.636,159.995
C00809=1021.713,385.981,348.921,172.612,49.636,159.993
C00810=1021.703,385.735,348.963,172.602,49.635,159.991
C00811=1021.694,385.488,349.006,172.593,49.635,159.990
C00812=1021.685,385.242,349.047,172.583,49.635,159.988
C00813=1021.676,384.995,349.089,172.573,49.635,159.987
C00814=1021.667,384.750,349.131,172.563,49.635,159.985
C00815=1021.658,384.503,349.173,172.554,49.634,159.983
C00816=1021.649,384.257,349.215,172.545,49.634,159.982
C00817=1021.639,384.011,349.256,172.535,49.634,159.980
C00818=1021.630,383.765,349.298,172.526,49.634,159.979
C00819=1021.621,383.518,349.339,172.516,49.634,159.977
C00820=1021.612,383.272,349.381,172.506,49.634,159.975
C00821=1021.604,383.026,349.423,172.496,49.634,159.974
C00822=1021.595,382.779,349.465,172.487,49.634,159.972
C00823=1021.585,382.533,349.506,172.477,49.634,159.971
C00824=1021.576,382.287,349.547,172.468,49.633,159.969
C00825=1021.567,382.040,349.589,172.459,49.634,159.968
C00826=1021.558,381.771,349.634,172.448,49.634,159.966
C00827=1021.548,381.501,349.679,172.438,49.633,159.964
C00828=1021.538,381.233,349.724,172.427,49.634,159.963
C00829=1021.529,380.963,349.770,172.418,49.634,159.961
C00830=1021.520,380.717,349.811,172.408,49.634,159.960
C00831=1021.511,380.470,349.853,172.398,49.633,159.958
C00832=1021.502,380.223,349.894,172.389,49.634,159.957
C00833=1021.493,379.978,349.935,172.380,49.634,159.955
C00834=1021.484,379.731,349.976,172.371,49.634,159.954
C00835=1021.475,379.485,350.017,172.361,49.634,159.952
C00836=1021.467,379.238,350.058,172.352,49.634,159.951
C00837=1021.458,378.992,350.100,172.343,49.634,159.949
C00838=1021.449,378.745,350.140,172.333,49.634,159.948
C00839=1021.441,378.500,350.182,172.324,49.634,159.946
C00840=1021.432,378.253,350.223,172.315,49.634,159.945
C00841=1021.423,378.006,350.264,172.306,49.635,159.943
C00842=1021.415,377.760,350.305,172.297,49.634,159.942
C00843=1021.407,377.513,350.346,172.288,49.635,159.941
C00844=1021.398,377.267,350.386,172.278,49.635,159.939
C00845=1021.389,377.021,350.428,172.270,49.635,159.938
C00846=1021.381,376.774,350.468,172.260,49.635,159.936
C00847=1021.372,376.527,350.509,172.252,49.635,159.935
C00848=1021.364,376.281,350.550,172.243,49.636,159.934
C00849=1021.355,376.035,350.590,172.233,49.636,159.932
C00850=1021.346,375.788,350.631,172.225,49.636,159.931
C00851=1021.337,375.542,350.671,172.216,49.637,159.930
C00852=1021.329,375.295,350.712,172.207,49.637,159.928
C00853=1021.320,375.049,350.752,172.198,49.637,159.927
C00854=1021.312,374.801,350.793,172.189,49.638,159.925
C00855=1021.303,374.555,350.833,172.180,49.638,159.924
C00856=1021.295,374.309,350.873,172.171,49.639,159.923
C00857=1021.286,374.062,350.914,172.162,49.639,159.921
C00858=1021.277,373.816,350.954,172.153,49.640,159.920
C00859=1021.268,373.568,350.994,172.145,49.640,159.919
C00860=1021.260,373.322,351.035,172.136,49.640,159.918
C00861=1021.252,373.076,351.075,172.127,49.640,159.916
C00862=1021.243,372.829,351.115,172.118,49.641,159.915
C00863=1021.235,372.583,351.155,172.110,49.641,159.914
C00864=1021.227,372.336,351.195,172.101,49.642,159.912
C00865=1021.218,372.090,351.235,172.092,49.643,159.911
C00866=1021.210,371.842,351.275,172.083,49.643,159.910
C00867=1021.201,371.596,351.315,172.075,49.643,159.908
C00868=1021.193,371.349,351.355,172.067,49.644,159.907
C00869=1021.184,371.103,351.395,172.058,49.645,159.906
C00870=1021.176,370.856,351.436,172.049,49.645,159.905
C00871=1021.168,370.609,351.475,172.040,49.645,159.903
C00872=1021.159,370.363,351.515,172.032,49.646,159.902
C00873=1021.151,370.116,351.555,172.023,49.647,159.901
C00874=1021.143,369.870,351.594,172.015,49.647,159.900
C00875=1021.135,369.623,351.635,172.006,49.648,159.899
C00876=1021.126,369.377,351.674,171.997,49.649,159.897
C00877=1021.119,369.130,351.714,171.989,49.649,159.896
C00878=1021.110,368.883,351.754,171.981,49.650,159.895
C00879=1021.102,368.636,351.794,171.972,49.651,159.894
C00880=1021.093,368.389,351.833,171.964,49.651,159.893
C00881=1021.085,368.143,351.874,171.956,49.652,159.891
C00882=1021.077,367.896,351.913,171.947,49.652,159.890
C00883=1021.069,367.649,351.952,171.938,49.653,159.889
C00884=1021.060,367.402,351.991,171.930,49.653,159.888
C00885=1021.053,367.155,352.031,171.921,49.654,159.887
C00886=1021.044,366.909,352.070,171.913,49.655,159.886
C00887=1021.036,366.662,352.109,171.905,49.656,159.884
C00888=1021.028,366.414,352.149,171.896,49.657,159.883
C00889=1021.019,366.167,352.188,171.888,49.658,159.882
C00890=1021.011,365.920,352.227,171.880,49.658,159.881
C00891=1021.003,365.674,352.266,171.872,49.659,159.880
C00892=1020.994,365.427,352.306,171.863,49.660,159.879
C00893=1020.986,365.180,352.344,171.855,49.661,159.878
C00894=1020.979,364.934,352.384,171.847,49.662,159.877
C00895=1020.971,364.686,352.422,171.839,49.663,159.875
C00896=1020.962,364.440,352.462,171.830,49.663,159.874
C00897=1020.954,364.193,352.500,171.822,49.664,159.873
C00898=1020.946,363.946,352.540,171.814,49.665,159.872
C00899=1020.937,363.699,352.578,171.807,49.666,159.871
C00900=1020.930,363.453,352.617,171.798,49.668,159.870
C00901=1020.922,363.205,352.657,171.790,49.668,159.869
C00902=1020.914,362.959,352.696,171.782,49.669,159.868
C00903=1020.906,362.712,352.734,171.774,49.670,159.867
C00904=1020.898,362.465,352.773,171.766,49.671,159.866
C00905=1020.890,362.218,352.812,171.758,49.672,159.865
C00906=1020.881,361.971,352.851,171.749,49.673,159.863
C00907=1020.874,361.725,352.889,171.741,49.674,159.862
C00908=1020.866,361.478,352.929,171.734,49.675,159.861
C00909=1020.858,361.231,352.967,171.726,49.676,159.861
C00910=1020.850,360.984,353.006,171.718,49.677,159.859
C00911=1020.842,360.737,353.044,171.710,49.678,159.858
C00912=1020.835,360.490,353.082,171.702,49.679,159.857
C00913=1020.826,360.244,353.122,171.695,49.680,159.856
C00914=1020.818,359.997,353.160,171.686,49.681,159.855
C00915=1020.811,359.750,353.199,171.678,49.683,159.854
C00916=1020.802,359.503,353.237,171.670,49.684,159.853
C00917=1020.795,359.256,353.276,171.662,49.685,159.852
C00918=1020.787,359.008,353.313,171.655,49.686,159.851
C00919=1020.779,358.762,353.352,171.647,49.687,159.850
C00920=1020.771,358.515,353.390,171.639,49.688,159.850
C00921=1020.764,358.268,353.428,171.631,49.689,159.849
C00922=1020.756,358.021,353.467,171.624,49.690,159.848
C00923=1020.748,357.774,353.505,171.616,49.691,159.847
C00924=1020.739,357.527,353.543,171.608,49.693,159.846
C00925=1020.732,357.280,353.581,171.600,49.694,159.845
C00926=1020.724,357.033,353.619,171.592,49.695,159.844
C00927=1020.717,356.786,353.657,171.584,49.697,159.843
C00928=1020.708,356.539,353.696,171.576,49.698,159.842
C00929=1020.701,356.292,353.734,171.569,49.699,159.841
C00930=1020.693,356.046,353.771,171.561,49.700,159.840
C00931=1020.685,355.798,353.809,171.554,49.702,159.839
C00932=1020.677,355.551,353.847,171.546,49.703,159.838
C00933=1020.669,355.304,353.886,171.538,49.704,159.837
C00934=1020.662,355.057,353.923,171.531,49.706,159.836
C00935=1020.654,354.811,353.961,171.523,49.707,159.835
C00936=1020.647,354.563,353.998,171.516,49.709,159.835
C00937=1020.638,354.316,354.037,171.508,49.710,159.834
C00938=1020.631,354.069,354.074,171.500,49.711,159.833
C00939=1020.623,353.822,354.111,171.493,49.713,159.832
C00940=1020.615,353.574,354.149,171.485,49.714,159.831
C00941=1020.608,353.328,354.187,171.477,49.715,159.830
C00942=1020.600,353.085,354.224,171.471,49.717,159.829
C00943=1020.592,352.841,354.261,171.463,49.718,159.829
C00944=1020.585,352.598,354.298,171.456,49.720,159.828
C00945=1020.578,352.354,354.335,171.448,49.721,159.827
C00946=1020.570,352.111,354.372,171.441,49.722,159.826
C00947=1020.562,351.868,354.409,171.433,49.724,159.825
C00948=1020.555,351.624,354.445,171.426,49.726,159.824
C00949=1020.546,351.381,354.482,171.419,49.727,159.824
C00950=1020.539,351.133,354.520,171.412,49.728,159.823
C00951=1020.532,350.886,354.558,171.404,49.730,159.822
C00952=1020.524,350.639,354.594,171.397,49.732,159.821
C00953=1020.517,350.392,354.632,171.389,49.733,159.820
C00954=1020.509,350.145,354.670,171.382,49.735,159.819
C00955=1020.502,349.898,354.706,171.375,49.736,159.819
C00956=1020.495,349.651,354.743,171.367,49.738,159.818
C00957=1020.487,349.404,354.780,171.360,49.740,159.817
C00958=1020.479,349.157,354.818,171.353,49.741,159.816
C00959=1020.472,348.910,354.855,171.346,49.742,159.815
C00960=1020.464,348.663,354.892,171.338,49.744,159.815
C00961=1020.457,348.415,354.929,171.331,49.746,159.814
C00962=1020.449,348.168,354.966,171.323,49.748,159.813
C00963=1020.442,347.921,355.003,171.316,49.749,159.812
C00964=1020.434,347.674,355.040,171.309,49.751,159.812
C00965=1020.427,347.426,355.077,171.302,49.752,159.811
C00966=1020.419,347.180,355.114,171.295,49.754,159.810
C00967=1020.412,346.932,355.151,171.287,49.756,159.809
C00968=1020.404,346.685,355.188,171.280,49.758,159.809
C00969=1020.396,346.438,355.224,171.273,49.760,159.808
C00970=1020.389,346.190,355.262,171.266,49.762,159.807
C00971=1020.381,345.943,355.298,171.258,49.763,159.806
C00972=1020.373,345.696,355.335,171.252,49.765,159.806
C00973=1020.367,345.448,355.372,171.245,49.767,159.805
C00974=1020.359,345.202,355.408,171.237,49.769,159.804
C00975=1020.352,344.955,355.444,171.230,49.771,159.804
C00976=1020.345,344.707,355.481,171.223,49.772,159.803
C00977=1020.337,344.460,355.518,171.217,49.774,159.802
C00978=1020.330,344.212,355.555,171.209,49.776,159.802
C00979=1020.323,343.966,355.591,171.202,49.778,159.801
C00980=1020.315,343.719,355.628,171.195,49.780,159.800
C00981=1020.308,343.471,355.665,171.187,49.782,159.799
C00982=1020.300,343.224,355.701,171.181,49.783,159.799
C00983=1020.293,342.977,355.737,171.174,49.786,159.798
C00984=1020.285,342.730,355.773,171.167,49.787,159.797
C00985=1020.278,342.482,355.810,171.160,49.790,159.797
C00986=1020.270,342.235,355.847,171.153,49.791,159.796
C00987=1020.263,341.988,355.882,171.146,49.793,159.796
C00988=1020.256,341.740,355.919,171.139,49.795,159.795
C00989=1020.249,341.493,355.955,171.132,49.797,159.794
C00990=1020.242,341.246,355.991,171.125,49.799,159.793
C00991=1020.234,340.999,356.027,171.118,49.801,159.793
C00992=1020.227,340.751,356.064,171.111,49.804,159.792
C00993=1020.220,340.504,356.100,171.104,49.805,159.792
C00994=1020.212,340.257,356.136,171.098,49.807,159.791
C00995=1020.205,340.009,356.172,171.091,49.809,159.790
C00996=1020.198,339.762,356.208,171.084,49.811,159.790
C00997=1020.191,339.515,356.244,171.076,49.814,159.789
C00998=1020.184,339.268,356.280,171.070,49.815,159.788
C00999=1020.176,339.020,356.317,171.063,49.817,159.788
C01000=1020.169,338.773,356.352,171.056,49.820,159.787
C01001=1020.162,338.525,356.388,171.050,49.822,159.787
C01002=1020.155,338.281,356.423,171.043,49.824,159.786
C01003=1020.147,338.036,356.459,171.036,49.826,159.786
C01004=1020.140,337.791,356.494,171.030,49.828,159.785
C01005=1020.133,337.546,356.530,171.023,49.830,159.784
C01006=1020.125,337.301,356.565,171.016,49.833,159.784
C01007=1020.118,337.056,356.600,171.010,49.835,159.783
C01008=1020.112,336.811,356.636,171.002,49.837,159.783
C01009=1020.104,336.566,356.672,170.995,49.839,159.782
C01010=1020.097,336.318,356.707,170.989,49.841,159.782
C01011=1020.090,336.071,356.743,170.982,49.844,159.781
C01012=1020.083,335.824,356.778,170.975,49.846,159.780
C01013=1020.076,335.576,356.813,170.969,49.848,159.780
C01014=1020.069,335.329,356.849,170.962,49.850,159.779
C01015=1020.062,335.081,356.885,170.955,49.853,159.779
C01016=1020.054,334.834,356.921,170.949,49.855,159.778
C01017=1020.047,334.587,356.956,170.942,49.857,159.778
C01018=1020.041,334.339,356.991,170.935,49.859,159.777
C01019=1020.033,334.092,357.027,170.930,49.862,159.777
C01020=1020.026,333.844,357.062,170.923,49.864,159.776
C01021=1020.019,333.597,357.098,170.916,49.867,159.776
C01022=1020.012,333.350,357.133,170.910,49.869,159.775
C01023=1020.005,333.102,357.169,170.903,49.871,159.775
C01024=1019.997,332.855,357.203,170.896,49.873,159.774
C01025=1019.991,332.608,357.239,170.890,49.876,159.774
C01026=1019.983,332.360,357.274,170.883,49.879,159.773
C01027=1019.977,332.112,357.309,170.877,49.881,159.773
C01028=1019.969,331.865,357.344,170.870,49.884,159.772
C01029=1019.962,331.618,357.379,170.863,49.886,159.772
C01030=1019.955,331.370,357.414,170.857,49.889,159.771
C01031=1019.948,331.123,357.449,170.850,49.891,159.771
C01032=1019.941,330.876,357.484,170.843,49.893,159.770
C01033=1019.934,330.628,357.519,170.838,49.896,159.770
C01034=1019.927,330.381,357.554,170.831,49.898,159.769
C01035=1019.920,330.133,357.589,170.825,49.901,159.769
C01036=1019.912,329.886,357.624,170.818,49.903,159.768
C01037=1019.905,329.638,357.659,170.811,49.906,159.768
C01038=1019.899,329.391,357.695,170.805,49.908,159.768
C01039=1019.891,329.143,357.728,170.799,49.911,159.767
C01040=1019.885,328.896,357.764,170.792,49.914,159.767
C01041=1019.878,328.649,357.799,170.786,49.916,159.766
C01042=1019.871,328.401,357.834,170.779,49.919,159.766
C01043=1019.864,328.154,357.868,170.773,49.921,159.765
C01044=1019.857,327.906,357.903,170.767,49.924,159.765
C01045=1019.850,327.659,357.938,170.761,49.926,159.765
C01046=1019.843,327.412,357.972,170.754,49.929,159.764
C01047=1019.836,327.164,358.007,170.747,49.932,159.764
C01048=1019.830,326.916,358.042,170.741,49.934,159.763
C01049=1019.823,326.669,358.077,170.735,49.937,159.763
C01050=1019.816,326.421,358.111,170.729,49.940,159.763
C01051=1019.808,326.174,358.146,170.722,49.942,159.762
C01052=1019.802,325.926,358.180,170.715,49.945,159.762
C01053=1019.795,325.679,358.214,170.710,49.948,159.761
C01054=1019.787,325.432,358.248,170.703,49.951,159.761
C01055=1019.780,325.184,358.282,170.697,49.954,159.761
C01056=1019.773,324.936,358.317,170.691,49.957,159.760
C01057=1019.766,324.689,358.351,170.684,49.960,159.760
C01058=1019.759,324.441,358.385,170.678,49.962,159.760
C01059=1019.752,324.193,358.419,170.672,49.965,159.759
C01060=1019.745,323.946,358.454,170.665,49.968,159.759
C01061=1019.738,323.699,358.488,170.660,49.971,159.759
C01062=1019.730,323.451,358.522,170.653,49.974,159.758
C01063=1019.723,323.205,358.556,170.647,49.977,159.758
C01064=1019.717,322.957,358.590,170.641,49.980,159.757
C01065=1019.710,322.709,358.624,170.635,49.982,159.757
C01066=1019.703,322.463,358.658,170.628,49.985,159.757
C01067=1019.696,322.215,358.692,170.622,49.988,159.756
C01068=1019.689,321.968,358.725,170.616,49.991,159.756
C01069=1019.682,321.720,358.759,170.610,49.995,159.756
C01070=1019.674,321.473,358.794,170.604,49.997,159.756
C01071=1019.668,321.226,358.828,170.597,50.000,159.755
C01072=1019.661,320.978,358.862,170.592,50.003,159.755
C01073=1019.654,320.731,358.895,170.585,50.006,159.755
C01074=1019.648,320.483,358.930,170.579,50.009,159.754
C01075=1019.641,320.236,358.963,170.573,50.012,159.754
C01076=1019.634,319.988,358.997,170.567,50.015,159.754
C01077=1019.627,319.740,359.031,170.561,50.018,159.753
C01078=1019.620,319.492,359.065,170.554,50.021,159.753
C01079=1019.614,319.245,359.098,170.549,50.024,159.753
C01080=1019.607,318.997,359.132,170.542,50.027,159.752
C01081=1019.599,318.749,359.166,170.537,50.030,159.752
C01082=1019.594,318.502,359.200,170.530,50.034,159.752
C01083=1019.586,318.254,359.234,170.525,50.036,159.752
C01084=1019.579,318.007,359.268,170.518,50.039,159.751
C01085=1019.573,317.760,359.301,170.513,50.043,159.751
C01086=1019.566,317.511,359.335,170.506,50.046,159.751
C01087=1019.560,317.264,359.368,170.500,50.048,159.750
C01088=1019.553,317.016,359.402,170.494,50.052,159.750
C01089=1019.545,316.769,359.436,170.489,50.055,159.750
C01090=1019.540,316.521,359.469,170.482,50.058,159.750
C01091=1019.533,316.273,359.503,170.477,50.061,159.750
C01092=1019.526,316.026,359.536,170.470,50.065,159.749
C01093=1019.519,315.778,359.570,170.465,50.067,159.749
C01094=1019.513,315.531,359.604,170.458,50.071,159.749
C01095=1019.506,315.283,359.637,170.453,50.074,159.749
C01096=1019.500,315.035,359.670,170.447,50.077,159.748
C01097=1019.493,314.788,359.704,170.441,50.080,159.748
C01098=1019.486,314.540,359.737,170.435,50.084,159.748
C01099=1019.480,314.292,359.771,170.429,50.086,159.748
C01100=1019.473,314.045,359.805,170.423,50.090,159.747
C01101=1019.466,313.797,359.838,170.417,50.093,159.747
C01102=1019.460,313.550,359.871,170.411,50.096,159.747
C01103=1019.454,313.301,359.905,170.405,50.100,159.747
C01104=1019.447,313.054,359.938,170.400,50.102,159.746
C01105=1019.441,312.807,359.971,170.394,50.106,159.746
C01106=1019.434,312.559,360.005,170.388,50.109,159.746
C01107=1019.428,312.311,360.038,170.382,50.112,159.746
C01108=1019.421,312.064,360.072,170.376,50.116,159.746
C01109=1019.415,311.816,360.105,170.370,50.119,159.745
C01110=1019.408,311.568,360.138,170.365,50.122,159.745
C01111=1019.402,311.321,360.171,170.358,50.126,159.745
C01112=1019.395,311.073,360.205,170.353,50.129,159.745
C01113=1019.389,310.825,360.237,170.348,50.132,159.745
C01114=1019.383,310.578,360.271,170.341,50.136,159.745
C01115=1019.376,310.330,360.304,170.336,50.138,159.744
C01116=1019.370,310.082,360.337,170.329,50.142,159.744
C01117=1019.364,309.835,360.371,170.324,50.145,159.744
C01118=1019.356,309.588,360.403,170.318,50.149,159.744
C01119=1019.350,309.339,360.436,170.313,50.152,159.744
C01120=1019.343,309.092,360.468,170.306,50.156,159.743
C01121=1019.337,308.844,360.500,170.301,50.159,159.743
C01122=1019.329,308.600,360.532,170.295,50.163,159.743
C01123=1019.323,308.355,360.565,170.289,50.166,159.743
C01124=1019.316,308.110,360.597,170.284,50.171,159.743
C01125=1019.310,307.865,360.630,170.278,50.174,159.743
C01126=1019.303,307.621,360.661,170.273,50.177,159.743
C01127=1019.296,307.376,360.694,170.267,50.181,159.743
C01128=1019.290,307.132,360.725,170.261,50.184,159.743
C01129=1019.283,306.888,360.757,170.255,50.188,159.742
C01130=1019.277,306.639,360.790,170.250,50.192,159.742
C01131=1019.270,306.391,360.823,170.244,50.196,159.742
C01132=1019.263,306.144,360.855,170.239,50.199,159.742
C01133=1019.257,305.896,360.888,170.233,50.203,159.742
C01134=1019.250,305.648,360.919,170.228,50.207,159.742
C01135=1019.244,305.401,360.952,170.221,50.210,159.742
C01136=1019.237,305.153,360.984,170.216,50.214,159.742
C01137=1019.230,304.905,361.017,170.210,50.217,159.741
C01138=1019.224,304.657,361.049,170.205,50.221,159.742
C01139=1019.217,304.410,361.081,170.199,50.225,159.741
C01140=1019.211,304.161,361.113,170.193,50.228,159.741
C01141=1019.204,303.914,361.145,170.187,50.233,159.741
C01142=1019.197,303.666,361.178,170.182,50.236,159.741
C01143=1019.191,303.418,361.210,170.176,50.240,159.741
C01144=1019.184,303.171,361.242,170.171,50.244,159.741
C01145=1019.178,302.923,361.274,170.165,50.247,159.741
C01146=1019.171,302.675,361.307,170.160,50.251,159.741
C01147=1019.165,302.427,361.339,170.154,50.255,159.741
C01148=1019.158,302.179,361.371,170.149,50.259,159.741
C01149=1019.152,301.931,361.403,170.142,50.263,159.741
C01150=1019.145,301.683,361.436,170.138,50.267,159.741
C01151=1019.139,301.436,361.467,170.132,50.270,159.741
C01152=1019.132,301.188,361.500,170.126,50.274,159.741
C01153=1019.126,300.940,361.531,170.121,50.278,159.741
C01154=1019.119,300.692,361.564,170.115,50.282,159.741
C01155=1019.113,300.445,361.595,170.110,50.285,159.740
C01156=1019.107,300.196,361.628,170.104,50.290,159.740
C01157=1019.100,299.949,361.660,170.099,50.293,159.740
C01158=1019.094,299.701,361.692,170.093,50.297,159.740
C01159=1019.088,299.453,361.723,170.088,50.301,159.740
C01160=1019.081,299.206,361.756,170.083,50.305,159.740
C01161=1019.075,298.958,361.788,170.077,50.309,159.740
C01162=1019.068,298.710,361.819,170.072,50.313,159.740
C01163=1019.062,298.462,361.852,170.066,50.317,159.740
C01164=1019.056,298.214,361.884,170.061,50.321,159.740
C01165=1019.049,297.966,361.915,170.055,50.325,159.740
C01166=1019.044,297.718,361.947,170.050,50.328,159.740
C01167=1019.037,297.470,361.979,170.044,50.333,159.740
C01168=1019.031,297.223,362.011,170.039,50.337,159.740
C01169=1019.024,296.975,362.042,170.034,50.340,159.740
C01170=1019.018,296.727,362.074,170.028,50.344,159.740
C01171=1019.012,296.479,362.106,170.023,50.348,159.740
C01172=1019.006,296.231,362.138,170.017,50.353,159.740
C01173=1019.000,295.984,362.170,170.012,50.356,159.740
C01174=1018.994,295.736,362.201,170.007,50.360,159.740
C01175=1018.987,295.488,362.234,170.001,50.364,159.740
C01176=1018.981,295.240,362.265,169.996,50.368,159.740
C01177=1018.975,294.992,362.297,169.990,50.373,159.740
C01178=1018.968,294.745,362.328,169.985,50.377,159.740
C01179=1018.962,294.496,362.360,169.979,50.380,159.740
C01180=1018.956,294.249,362.392,169.974,50.384,159.740
C01181=1018.950,294.000,362.424,169.969,50.388,159.740
C01182=1018.944,293.765,362.453,169.964,50.392,159.740
C01183=1018.939,293.529,362.483,169.960,50.396,159.740
C01184=1018.932,293.293,362.514,169.954,50.401,159.740
C01185=1018.927,293.057,362.544,169.948,50.404,159.740
C01186=1018.921,292.821,362.573,169.943,50.408,159.740
C01187=1018.915,292.585,362.603,169.939,50.412,159.740
C01188=1018.908,292.350,362.633,169.934,50.416,159.741
C01189=1018.903,292.114,362.663,169.929,50.420,159.741
C01190=1018.896,291.866,362.693,169.923,50.425,159.741
C01191=1018.890,291.618,362.725,169.918,50.429,159.741
C01192=1018.884,291.371,362.757,169.913,50.434,159.741
C01193=1018.878,291.123,362.788,169.908,50.438,159.741
C01194=1018.871,290.874,362.819,169.902,50.442,159.741
C01195=1018.865,290.627,362.850,169.897,50.446,159.741
C01196=1018.859,290.378,362.881,169.891,50.450,159.741
C01197=1018.852,290.130,362.912,169.887,50.455,159.741
C01198=1018.846,289.883,362.942,169.881,50.459,159.741
C01199=1018.839,289.635,362.974,169.876,50.463,159.741
C01200=1018.833,289.386,363.004,169.871,50.467,159.742
C01201=1018.827,289.139,363.036,169.865,50.472,159.742
C01202=1018.820,288.890,363.066,169.861,50.476,159.742
C01203=1018.814,288.642,363.098,169.855,50.481,159.742
C01204=1018.809,288.394,363.129,169.850,50.485,159.742
C01205=1018.802,288.147,363.160,169.844,50.490,159.742
C01206=1018.796,287.899,363.190,169.839,50.494,159.742
C01207=1018.789,287.651,363.222,169.834,50.499,159.742
C01208=1018.784,287.403,363.252,169.829,50.503,159.742
C01209=1018.777,287.154,363.283,169.824,50.508,159.743
C01210=1018.771,286.907,363.314,169.819,50.512,159.743
C01211=1018.765,286.659,363.345,169.813,50.517,159.743
C01212=1018.758,286.410,363.375,169.808,50.521,159.743
C01213=1018.752,286.163,363.406,169.803,50.526,159.743
C01214=1018.746,285.914,363.437,169.798,50.530,159.743
C01215=1018.740,285.667,363.468,169.792,50.535,159.743
C01216=1018.733,285.418,363.498,169.788,50.539,159.744
C01217=1018.727,285.171,363.529,169.783,50.544,159.744
C01218=1018.721,284.922,363.560,169.777,50.548,159.744
C01219=1018.715,284.675,363.590,169.773,50.553,159.744
C01220=1018.708,284.427,363.620,169.767,50.557,159.744
C01221=1018.702,284.179,363.651,169.762,50.562,159.744
C01222=1018.696,283.931,363.681,169.757,50.567,159.745
C01223=1018.690,283.682,363.712,169.752,50.571,159.745
C01224=1018.683,283.435,363.742,169.747,50.576,159.745
C01225=1018.677,283.186,363.772,169.741,50.581,159.745
C01226=1018.671,282.938,363.803,169.736,50.585,159.745
C01227=1018.665,282.690,363.833,169.731,50.590,159.745
C01228=1018.659,282.442,363.864,169.726,50.595,159.746
C01229=1018.652,282.195,363.894,169.721,50.600,159.746
C01230=1018.646,281.946,363.924,169.716,50.604,159.746
C01231=1018.640,281.698,363.955,169.710,50.609,159.746
C01232=1018.634,281.450,363.985,169.706,50.614,159.746
C01233=1018.627,281.202,364.015,169.700,50.619,159.747
C01234=1018.621,280.954,364.045,169.696,50.623,159.747
C01235=1018.615,280.706,364.076,169.690,50.628,159.747
C01236=1018.609,280.458,364.107,169.686,50.632,159.747
C01237=1018.602,280.210,364.136,169.680,50.637,159.747
C01238=1018.596,279.961,364.166,169.676,50.642,159.748
C01239=1018.591,279.713,364.197,169.670,50.647,159.748
C01240=1018.585,279.466,364.227,169.666,50.652,159.748
C01241=1018.578,279.217,364.257,169.660,50.657,159.748
C01242=1018.572,278.987,364.285,169.655,50.661,159.748
C01243=1018.566,278.758,364.313,169.651,50.666,159.749
C01244=1018.561,278.529,364.341,169.646,50.670,159.749
C01245=1018.555,278.299,364.368,169.641,50.674,159.749
C01246=1018.550,278.069,364.397,169.637,50.679,159.749
C01247=1018.544,277.839,364.424,169.632,50.684,159.750
C01248=1018.539,277.610,364.452,169.628,50.688,159.750
C01249=1018.533,277.380,364.480,169.623,50.693,159.750
C01250=1018.527,277.132,364.510,169.619,50.697,159.750
C01251=1018.520,276.884,364.540,169.613,50.702,159.750
C01252=1018.515,276.636,364.570,169.609,50.707,159.751
C01253=1018.509,276.388,364.600,169.603,50.712,159.751
C01254=1018.503,276.140,364.629,169.599,50.717,159.751
C01255=1018.496,275.891,364.660,169.593,50.722,159.751
C01256=1018.490,275.643,364.689,169.589,50.727,159.752
C01257=1018.484,275.395,364.719,169.584,50.732,159.752
C01258=1018.478,275.147,364.749,169.579,50.737,159.752
C01259=1018.472,274.899,364.779,169.574,50.742,159.752
C01260=1018.465,274.650,364.808,169.569,50.747,159.753
C01261=1018.460,274.402,364.839,169.564,50.752,159.753
C01262=1018.453,274.154,364.868,169.560,50.757,159.753
C01263=1018.448,273.906,364.897,169.554,50.762,159.754
C01264=1018.441,273.658,364.927,169.549,50.767,159.754
C01265=1018.436,273.410,364.957,169.545,50.773,159.754
C01266=1018.429,273.162,364.987,169.539,50.778,159.754
C01267=1018.423,272.913,365.016,169.535,50.782,159.755
C01268=1018.417,272.665,365.045,169.530,50.788,159.755
C01269=1018.411,272.417,365.076,169.525,50.793,159.755
C01270=1018.405,272.169,365.105,169.520,50.798,159.756
C01271=1018.399,271.921,365.135,169.516,50.803,159.756
C01272=1018.393,271.673,365.164,169.510,50.808,159.756
C01273=1018.386,271.425,365.193,169.506,50.813,159.756
C01274=1018.381,271.177,365.223,169.501,50.819,159.757
C01275=1018.375,270.929,365.252,169.495,50.824,159.757
C01276=1018.369,270.680,365.282,169.491,50.829,159.758
C01277=1018.363,270.432,365.311,169.486,50.834,159.758
C01278=1018.356,270.184,365.341,169.482,50.840,159.758
C01279=1018.350,269.935,365.370,169.476,50.845,159.758
C01280=1018.344,269.687,365.399,169.472,50.850,159.759
C01281=1018.338,269.439,365.429,169.467,50.855,159.759
C01282=1018.332,269.191,365.458,169.462,50.861,159.760
C01283=1018.326,268.942,365.487,169.457,50.866,159.760
C01284=1018.320,268.694,365.517,169.452,50.872,159.760
C01285=1018.314,268.446,365.546,169.447,50.876,159.760
C01286=1018.308,268.198,365.575,169.442,50.882,159.761
C01287=1018.302,267.950,365.604,169.438,50.887,159.761
C01288=1018.295,267.702,365.633,169.433,50.893,159.761
C01289=1018.290,267.453,365.663,169.428,50.898,159.762
C01290=1018.284,267.205,365.692,169.423,50.903,159.762
C01291=1018.277,266.957,365.721,169.418,50.909,159.762
C01292=1018.272,266.709,365.749,169.414,50.914,159.763
C01293=1018.266,266.461,365.779,169.409,50.920,159.763
C01294=1018.260,266.213,365.808,169.404,50.925,159.764
C01295=1018.254,265.965,365.837,169.400,50.930,159.764
C01296=1018.248,265.716,365.865,169.395,50.936,159.764
C01297=1018.242,265.468,365.894,169.390,50.941,159.765
C01298=1018.236,265.219,365.924,169.385,50.947,159.765
C01299=1018.230,264.971,365.953,169.380,50.952,159.765
C01300=1018.224,264.723,365.982,169.376,50.958,159.766
C01301=1018.218,264.474,366.010,169.371,50.964,159.766
C01302=1018.212,264.247,366.037,169.366,50.968,159.767
C01303=1018.207,264.020,366.063,169.362,50.974,159.767
C01304=1018.201,263.793,366.090,169.358,50.978,159.767
C01305=1018.196,263.565,366.116,169.354,50.984,159.768
C01306=1018.190,263.338,366.143,169.349,50.989,159.768
C01307=1018.185,263.110,366.170,169.345,50.994,159.769
C01308=1018.179,262.883,366.196,169.341,50.999,159.769
C01309=1018.173,262.655,366.221,169.337,51.004,159.769
C01310=1018.167,262.408,366.250,169.332,51.010,159.770
C01311=1018.162,262.159,366.280,169.326,51.015,159.770
C01312=1018.156,261.910,366.308,169.322,51.021,159.770
C01313=1018.150,261.662,366.337,169.317,51.026,159.771
C01314=1018.144,261.413,366.365,169.313,51.032,159.771
C01315=1018.138,261.166,366.394,169.308,51.037,159.772
C01316=1018.132,260.918,366.423,169.303,51.043,159.772
C01317=1018.126,260.669,366.451,169.299,51.049,159.772
C01318=1018.120,260.421,366.481,169.294,51.054,159.773
C01319=1018.114,260.172,366.509,169.289,51.061,159.773
C01320=1018.108,259.925,366.538,169.285,51.066,159.774
C01321=1018.102,259.676,366.566,169.280,51.072,159.774
C01322=1018.095,259.428,366.594,169.275,51.078,159.775
C01323=1018.089,259.180,366.623,169.271,51.083,159.775
C01324=1018.084,258.931,366.651,169.266,51.090,159.776
C01325=1018.077,258.683,366.678,169.261,51.096,159.776
C01326=1018.071,258.434,366.707,169.256,51.101,159.777
C01327=1018.065,258.186,366.736,169.252,51.107,159.777
C01328=1018.058,257.938,366.763,169.248,51.113,159.778
C01329=1018.053,257.690,366.791,169.243,51.119,159.778
C01330=1018.047,257.441,366.820,169.237,51.125,159.778
C01331=1018.040,257.192,366.847,169.234,51.131,159.779
C01332=1018.034,256.944,366.876,169.229,51.137,159.779
C01333=1018.029,256.696,366.904,169.224,51.142,159.780
C01334=1018.022,256.448,366.932,169.219,51.149,159.780
C01335=1018.016,256.199,366.960,169.215,51.154,159.781
C01336=1018.010,255.951,366.988,169.210,51.161,159.782
C01337=1018.004,255.703,367.016,169.205,51.167,159.782
C01338=1017.998,255.454,367.044,169.200,51.172,159.782
C01339=1017.992,255.206,367.072,169.197,51.178,159.783
C01340=1017.986,254.958,367.101,169.192,51.184,159.783
C01341=1017.980,254.709,367.129,169.187,51.191,159.784
C01342=1017.974,254.461,367.157,169.182,51.197,159.784
C01343=1017.968,254.213,367.185,169.178,51.203,159.785
C01344=1017.962,253.964,367.213,169.173,51.208,159.785
C01345=1017.956,253.716,367.241,169.169,51.215,159.786
C01346=1017.950,253.467,367.269,169.164,51.221,159.786
C01347=1017.944,253.219,367.297,169.160,51.227,159.787
C01348=1017.938,252.971,367.325,169.155,51.233,159.787
C01349=1017.932,252.722,367.353,169.150,51.239,159.788
C01350=1017.926,252.474,367.380,169.145,51.245,159.788
C01351=1017.920,252.226,367.409,169.142,51.251,159.789
C01352=1017.915,251.978,367.437,169.137,51.258,159.790
C01353=1017.908,251.729,367.464,169.132,51.263,159.790
C01354=1017.902,251.480,367.492,169.127,51.270,159.791
C01355=1017.897,251.232,367.520,169.123,51.275,159.791
C01356=1017.890,250.983,367.548,169.119,51.282,159.792
C01357=1017.885,250.735,367.576,169.114,51.288,159.792
C01358=1017.878,250.487,367.603,169.109,51.294,159.793
C01359=1017.873,250.239,367.631,169.105,51.300,159.793
C01360=1017.867,249.990,367.660,169.101,51.307,159.794
C01361=1017.861,249.742,367.686,169.096,51.313,159.794
C01362=1017.856,249.513,367.712,169.092,51.319,159.795
C01363=1017.851,249.286,367.738,169.088,51.324,159.795
C01364=1017.845,249.058,367.764,169.083,51.330,159.796
C01365=1017.840,248.829,367.788,169.079,51.335,159.796
C01366=1017.835,248.601,367.815,169.076,51.342,159.797
C01367=1017.828,248.372,367.840,169.072,51.347,159.797
C01368=1017.823,248.144,367.865,169.067,51.352,159.798
C01369=1017.818,247.915,367.891,169.062,51.358,159.798
C01370=1017.812,247.668,367.919,169.059,51.364,159.799
C01371=1017.807,247.419,367.946,169.054,51.371,159.800
C01372=1017.800,247.170,367.974,169.050,51.377,159.800
C01373=1017.795,246.922,368.002,169.045,51.384,159.801
C01374=1017.789,246.673,368.029,169.041,51.389,159.801
C01375=1017.783,246.425,368.057,169.036,51.396,159.802
C01376=1017.777,246.177,368.085,169.032,51.402,159.802
C01377=1017.772,245.928,368.112,169.027,51.409,159.803
C01378=1017.766,245.680,368.140,169.023,51.415,159.804
C01379=1017.760,245.431,368.168,169.019,51.422,159.804
C01380=1017.755,245.183,368.195,169.014,51.427,159.805
C01381=1017.749,244.935,368.223,169.009,51.434,159.805
C01382=1017.744,244.686,368.250,169.005,51.440,159.806
C01383=1017.737,244.438,368.278,169.001,51.447,159.806
C01384=1017.732,244.190,368.306,168.996,51.453,159.807
C01385=1017.726,243.940,368.333,168.992,51.460,159.808
C01386=1017.720,243.693,368.361,168.987,51.466,159.808
C01387=1017.715,243.444,368.388,168.983,51.473,159.809
C01388=1017.709,243.196,368.415,168.979,51.479,159.810
C01389=1017.704,242.947,368.443,168.974,51.485,159.810
C01390=1017.698,242.699,368.470,168.970,51.492,159.811
C01391=1017.691,242.450,368.497,168.965,51.498,159.811
C01392=1017.686,242.201,368.524,168.961,51.505,159.812
C01393=1017.680,241.954,368.552,168.956,51.511,159.812
C01394=1017.674,241.705,368.579,168.952,51.519,159.813
C01395=1017.668,241.457,368.607,168.948,51.525,159.814
C01396=1017.663,241.208,368.633,168.944,51.531,159.815
C01397=1017.657,240.960,368.660,168.939,51.538,159.815
C01398=1017.651,240.710,368.688,168.935,51.544,159.816
C01399=1017.645,240.463,368.715,168.930,51.551,159.816
C01400=1017.639,240.214,368.742,168.926,51.558,159.817
C01401=1017.634,239.966,368.769,168.921,51.565,159.818
C01402=1017.628,239.717,368.797,168.917,51.571,159.818
C01403=1017.622,239.469,368.823,168.912,51.578,159.819
C01404=1017.617,239.220,368.850,168.909,51.585,159.820
C01405=1017.611,238.972,368.877,168.904,51.591,159.820
C01406=1017.605,238.723,368.904,168.900,51.598,159.821
C01407=1017.599,238.475,368.932,168.895,51.605,159.822
C01408=1017.593,238.227,368.958,168.891,51.611,159.822
C01409=1017.587,237.978,368.985,168.887,51.619,159.823
C01410=1017.581,237.730,369.011,168.882,51.625,159.824
C01411=1017.575,237.481,369.038,168.878,51.632,159.824
C01412=1017.569,237.233,369.065,168.873,51.639,159.825
C01413=1017.563,236.984,369.092,168.869,51.645,159.826
C01414=1017.558,236.736,369.119,168.865,51.653,159.826
C01415=1017.553,236.487,369.146,168.860,51.659,159.827
C01416=1017.546,236.238,369.173,168.856,51.666,159.828
C01417=1017.540,235.990,369.199,168.851,51.673,159.828
C01418=1017.535,235.741,369.226,168.847,51.680,159.829
C01419=1017.529,235.493,369.253,168.843,51.687,159.830
C01420=1017.523,235.245,369.279,168.838,51.694,159.831
C01421=1017.517,234.996,369.306,168.834,51.701,159.831
C01422=1017.512,234.765,369.331,168.831,51.707,159.832
C01423=1017.506,234.533,369.355,168.826,51.714,159.833
C01424=1017.500,234.301,369.380,168.823,51.720,159.833
C01425=1017.495,234.070,369.405,168.818,51.727,159.834
C01426=1017.490,233.838,369.429,168.813,51.733,159.834
C01427=1017.485,233.607,369.454,168.810,51.740,159.835
C01428=1017.479,233.374,369.479,168.806,51.747,159.836
C01429=1017.474,233.143,369.504,168.802,51.753,159.837
C01430=1017.467,232.895,369.530,168.798,51.760,159.837
C01431=1017.462,232.646,369.557,168.793,51.767,159.838
C01432=1017.456,232.397,369.583,168.789,51.774,159.839
C01433=1017.450,232.149,369.609,168.785,51.781,159.840
C01434=1017.445,231.901,369.636,168.781,51.788,159.840
C01435=1017.439,231.652,369.663,168.776,51.795,159.841
C01436=1017.433,231.404,369.689,168.772,51.802,159.842
C01437=1017.427,231.155,369.715,168.768,51.810,159.843
C01438=1017.422,230.907,369.742,168.764,51.816,159.843
C01439=1017.416,230.658,369.768,168.759,51.823,159.844
C01440=1017.410,230.409,369.794,168.755,51.831,159.845
C01441=1017.405,230.161,369.821,168.751,51.838,159.845
C01442=1017.399,229.913,369.848,168.746,51.846,159.846
C01443=1017.393,229.664,369.874,168.741,51.852,159.847
C01444=1017.388,229.415,369.900,168.737,51.859,159.848
C01445=1017.382,229.167,369.927,168.733,51.867,159.848
C01446=1017.376,228.918,369.952,168.729,51.874,159.849
C01447=1017.370,228.670,369.979,168.725,51.881,159.850
C01448=1017.364,228.421,370.005,168.721,51.888,159.851
C01449=1017.359,228.172,370.032,168.717,51.896,159.852
C01450=1017.353,227.923,370.057,168.712,51.903,159.852
C01451=1017.347,227.675,370.084,168.708,51.910,159.853
C01452=1017.341,227.427,370.110,168.704,51.918,159.854
C01453=1017.335,227.178,370.136,168.699,51.925,159.855
C01454=1017.330,226.930,370.163,168.695,51.932,159.855
C01455=1017.324,226.681,370.189,168.691,51.940,159.856
C01456=1017.319,226.432,370.215,168.687,51.947,159.857
C01457=1017.312,226.184,370.241,168.683,51.954,159.858
C01458=1017.307,225.935,370.267,168.678,51.962,159.859
C01459=1017.300,225.687,370.293,168.673,51.969,159.859
C01460=1017.295,225.438,370.319,168.670,51.977,159.860
C01461=1017.289,225.189,370.345,168.666,51.984,159.861
C01462=1017.284,224.941,370.369,168.661,51.992,159.862
C01463=1017.278,224.692,370.396,168.657,51.999,159.863
C01464=1017.272,224.444,370.421,168.653,52.006,159.863
C01465=1017.266,224.195,370.447,168.649,52.015,159.864
C01466=1017.260,223.947,370.473,168.644,52.022,159.865
C01467=1017.254,223.698,370.499,168.640,52.029,159.866
C01468=1017.249,223.449,370.525,168.636,52.036,159.867
C01469=1017.243,223.200,370.551,168.631,52.045,159.868
C01470=1017.237,222.952,370.577,168.627,52.052,159.868
C01471=1017.231,222.704,370.602,168.623,52.059,159.869
C01472=1017.226,222.455,370.628,168.619,52.067,159.870
C01473=1017.220,222.206,370.654,168.616,52.075,159.871
C01474=1017.214,221.957,370.679,168.610,52.082,159.872
C01475=1017.209,221.708,370.705,168.606,52.090,159.873
C01476=1017.202,221.460,370.731,168.603,52.098,159.874
C01477=1017.197,221.212,370.757,168.599,52.105,159.874
C01478=1017.191,220.963,370.782,168.594,52.113,159.875
C01479=1017.186,220.714,370.808,168.590,52.121,159.876
C01480=1017.179,220.465,370.834,168.586,52.128,159.877
C01481=1017.174,220.216,370.860,168.582,52.136,159.878
C01482=1017.169,219.981,370.884,168.578,52.143,159.879
C01483=1017.163,219.745,370.909,168.574,52.151,159.879
C01484=1017.158,219.510,370.933,168.570,52.158,159.880
C01485=1017.153,219.274,370.957,168.566,52.165,159.881
C01486=1017.147,219.039,370.981,168.562,52.172,159.882
C01487=1017.142,218.803,371.005,168.557,52.180,159.883
C01488=1017.136,218.567,371.029,168.553,52.187,159.883
C01489=1017.131,218.331,371.054,168.550,52.194,159.884
C01490=1017.125,218.082,371.080,168.546,52.202,159.885
C01491=1017.120,217.834,371.105,168.542,52.210,159.886
C01492=1017.114,217.585,371.130,168.538,52.218,159.887
C01493=1017.107,217.337,371.155,168.533,52.226,159.888
C01494=1017.102,217.088,371.181,168.529,52.233,159.889
C01495=1017.096,216.840,371.206,168.526,52.241,159.890
C01496=1017.090,216.591,371.232,168.521,52.250,159.891
C01497=1017.085,216.341,371.257,168.517,52.257,159.891
C01498=1017.079,216.093,371.282,168.512,52.266,159.892
C01499=1017.073,215.845,371.307,168.509,52.274,159.893
C01500=1017.067,215.596,371.332,168.504,52.281,159.894
C01501=1017.061,215.347,371.358,168.500,52.289,159.895
C01502=1017.056,215.099,371.383,168.496,52.297,159.896
C01503=1017.050,214.850,371.408,168.491,52.306,159.897
C01504=1017.044,214.601,371.433,168.488,52.314,159.898
C01505=1017.039,214.353,371.459,168.484,52.321,159.899
C01506=1017.033,214.104,371.483,168.479,52.329,159.900
C01507=1017.027,213.855,371.509,168.476,52.337,159.901
C01508=1017.021,213.607,371.534,168.471,52.346,159.902
C01509=1017.016,213.358,371.560,168.467,52.354,159.903
C01510=1017.010,213.109,371.584,168.463,52.361,159.903
C01511=1017.004,212.861,371.609,168.459,52.370,159.904
C01512=1016.998,212.612,371.635,168.455,52.378,159.905
C01513=1016.993,212.363,371.659,168.450,52.386,159.906
C01514=1016.987,212.115,371.685,168.447,52.394,159.907
C01515=1016.981,211.866,371.710,168.443,52.402,159.908
C01516=1016.976,211.617,371.734,168.438,52.411,159.909
C01517=1016.970,211.368,371.760,168.435,52.419,159.910
C01518=1016.965,211.120,371.785,168.430,52.427,159.911
C01519=1016.959,210.871,371.810,168.427,52.435,159.912
C01520=1016.953,210.622,371.835,168.422,52.443,159.913
C01521=1016.948,210.374,371.860,168.418,52.451,159.914
C01522=1016.942,210.125,371.885,168.413,52.459,159.915
C01523=1016.936,209.877,371.910,168.410,52.467,159.916
C01524=1016.930,209.628,371.935,168.405,52.476,159.917
C01525=1016.925,209.380,371.960,168.402,52.484,159.918
C01526=1016.920,209.130,371.985,168.397,52.493,159.919
C01527=1016.914,208.882,372.010,168.394,52.501,159.920
C01528=1016.908,208.633,372.035,168.389,52.509,159.921
C01529=1016.903,208.384,372.059,168.386,52.517,159.922
C01530=1016.896,208.136,372.084,168.381,52.526,159.923
C01531=1016.891,207.887,372.109,168.377,52.534,159.924
C01532=1016.885,207.638,372.134,168.373,52.542,159.925
C01533=1016.880,207.390,372.158,168.370,52.551,159.926
C01534=1016.873,207.141,372.184,168.365,52.560,159.927
C01535=1016.868,206.892,372.208,168.361,52.568,159.928
C01536=1016.862,206.643,372.233,168.357,52.576,159.929
C01537=1016.857,206.395,372.257,168.353,52.585,159.930
C01538=1016.851,206.146,372.282,168.349,52.593,159.931
C01539=1016.845,205.897,372.306,168.344,52.602,159.932
C01540=1016.839,205.649,372.332,168.341,52.610,159.933
C01541=1016.834,205.400,372.356,168.337,52.619,159.934
C01542=1016.828,205.161,372.380,168.333,52.627,159.935
C01543=1016.823,204.924,372.403,168.329,52.635,159.936
C01544=1016.817,204.685,372.426,168.325,52.643,159.937
C01545=1016.812,204.447,372.450,168.321,52.652,159.938
C01546=1016.806,204.209,372.473,168.317,52.660,159.939
C01547=1016.800,203.971,372.496,168.313,52.668,159.940
C01548=1016.795,203.733,372.520,168.310,52.676,159.941
C01549=1016.770,202.498,372.635,167.815,52.600,159.826
C01550=1016.766,202.249,372.658,167.810,52.611,159.827
C01551=1016.762,202.000,372.680,167.805,52.620,159.828
C01552=1016.757,201.752,372.703,167.801,52.630,159.829
C01553=1016.752,201.503,372.726,167.796,52.640,159.830
C01554=1016.747,201.254,372.748,167.791,52.650,159.831
C01555=1016.742,201.006,372.771,167.787,52.659,159.832
C01556=1016.738,200.756,372.794,167.782,52.669,159.833
C01557=1016.733,200.508,372.817,167.777,52.679,159.834
C01558=1016.729,200.258,372.839,167.773,52.689,159.836
C01559=1016.724,200.010,372.863,167.768,52.698,159.836
C01560=1016.719,199.760,372.885,167.764,52.708,159.838
C01561=1016.714,199.512,372.908,167.759,52.718,159.839
C01562=1016.710,199.263,372.930,167.754,52.728,159.840
C01563=1016.705,199.013,372.953,167.750,52.737,159.841
C01564=1016.700,198.765,372.976,167.745,52.747,159.842
C01565=1016.696,198.516,372.998,167.741,52.758,159.843
C01566=1016.690,198.266,373.020,167.736,52.767,159.844
C01567=1016.686,198.018,373.043,167.732,52.777,159.845
C01568=1016.681,197.769,373.065,167.727,52.787,159.847
C01569=1016.676,197.520,373.087,167.722,52.798,159.848
C01570=1016.671,197.270,373.110,167.718,52.807,159.849
C01571=1016.667,197.022,373.131,167.713,52.817,159.850
C01572=1016.661,196.773,373.154,167.708,52.827,159.851
C01573=1016.657,196.525,373.176,167.704,52.837,159.852
C01574=1016.652,196.275,373.199,167.699,52.847,159.853
C01575=1016.647,196.026,373.221,167.695,52.857,159.855
C01576=1016.642,195.777,373.242,167.691,52.867,159.856
C01577=1016.638,195.528,373.265,167.686,52.877,159.857
C01578=1016.633,195.280,373.288,167.681,52.887,159.858
C01579=1016.628,195.030,373.310,167.677,52.897,159.859
C01580=1016.623,194.781,373.332,167.672,52.907,159.860
C01581=1016.619,194.532,373.354,167.668,52.916,159.861
C01582=1016.614,194.284,373.376,167.664,52.927,159.863
C01583=1016.609,194.035,373.398,167.659,52.937,159.864
C01584=1016.605,193.786,373.420,167.655,52.946,159.865
C01585=1016.600,193.536,373.442,167.650,52.957,159.866
C01586=1016.595,193.287,373.464,167.646,52.967,159.867
C01587=1016.591,193.038,373.487,167.642,52.977,159.868
C01588=1016.586,192.789,373.509,167.636,52.986,159.869
C01589=1016.581,192.541,373.531,167.633,52.996,159.871
C01590=1016.576,192.292,373.552,167.628,53.007,159.872
C01591=1016.572,192.043,373.575,167.624,53.017,159.873
C01592=1016.567,191.793,373.597,167.619,53.026,159.874
C01593=1016.562,191.544,373.619,167.614,53.037,159.875
C01594=1016.558,191.295,373.641,167.611,53.047,159.877
C01595=1016.553,191.046,373.663,167.606,53.056,159.877
C01596=1016.548,190.797,373.685,167.602,53.066,159.879
C01597=1016.543,190.549,373.707,167.597,53.077,159.880
C01598=1016.539,190.300,373.729,167.593,53.086,159.881
C01599=1016.534,190.051,373.751,167.588,53.096,159.882
C01600=1016.530,189.802,373.773,167.585,53.106,159.883
C01601=1016.526,189.553,373.796,167.580,53.116,159.885
C01602=1016.521,189.304,373.818,167.576,53.126,159.886
C01603=1016.516,189.055,373.839,167.571,53.136,159.887
C01604=1016.511,188.806,373.861,167.567,53.146,159.888
C01605=1016.507,188.557,373.883,167.563,53.156,159.889
C01606=1016.502,188.308,373.905,167.559,53.166,159.890
C01607=1016.498,188.059,373.927,167.554,53.176,159.891
C01608=1016.493,187.810,373.949,167.550,53.186,159.893
C01609=1016.489,187.561,373.971,167.546,53.196,159.894
C01610=1016.483,187.280,373.995,167.541,53.207,159.895
C01611=1016.478,187.001,374.020,167.536,53.218,159.896
C01612=1016.473,186.720,374.045,167.532,53.229,159.898
C01613=1016.468,186.440,374.069,167.526,53.241,159.899
C01614=1016.463,186.191,374.091,167.523,53.251,159.900
C01615=1016.459,185.942,374.113,167.518,53.261,159.901
C01616=1016.454,185.693,374.135,167.514,53.270,159.903
C01617=1016.450,185.445,374.157,167.509,53.281,159.904
C01618=1016.445,185.195,374.178,167.506,53.291,159.905
C01619=1016.441,184.946,374.201,167.501,53.301,159.906
C01620=1016.436,184.697,374.222,167.497,53.310,159.907
C01621=1016.432,184.448,374.244,167.493,53.320,159.909
C01622=1016.427,184.200,374.265,167.489,53.331,159.910
C01623=1016.423,183.951,374.288,167.484,53.340,159.911
C01624=1016.419,183.702,374.309,167.480,53.351,159.912
C01625=1016.414,183.452,374.331,167.476,53.361,159.913
C01626=1016.410,183.203,374.353,167.473,53.371,159.914
C01627=1016.405,182.954,374.375,167.468,53.380,159.915
C01628=1016.401,182.705,374.396,167.464,53.390,159.917
C01629=1016.396,182.456,374.418,167.459,53.401,159.918
C01630=1016.392,182.206,374.440,167.455,53.410,159.919
C01631=1016.387,181.957,374.462,167.452,53.420,159.920
C01632=1016.383,181.709,374.482,167.447,53.430,159.921
C01633=1016.378,181.460,374.504,167.443,53.440,159.923
C01634=1016.373,181.211,374.525,167.439,53.451,159.924
C01635=1016.369,180.961,374.546,167.435,53.461,159.925
C01636=1016.364,180.713,374.568,167.431,53.471,159.926
C01637=1016.359,180.463,374.588,167.427,53.481,159.928
C01638=1016.354,180.214,374.609,167.422,53.492,159.929
C01639=1016.350,179.965,374.631,167.418,53.502,159.930
C01640=1016.345,179.717,374.651,167.414,53.512,159.931
C01641=1016.340,179.467,374.673,167.410,53.523,159.932
C01642=1016.335,179.218,374.693,167.406,53.533,159.934
C01643=1016.330,178.969,374.714,167.401,53.543,159.935
C01644=1016.326,178.719,374.735,167.398,53.553,159.936
C01645=1016.320,178.471,374.757,167.393,53.564,159.937
C01646=1016.316,178.222,374.778,167.390,53.574,159.939
C01647=1016.312,177.973,374.799,167.386,53.585,159.940
C01648=1016.307,177.724,374.819,167.382,53.595,159.941
C01649=1016.302,177.474,374.840,167.377,53.605,159.943
C01650=1016.297,177.225,374.861,167.374,53.615,159.944
C01651=1016.293,176.977,374.882,167.369,53.626,159.945
C01652=1016.288,176.727,374.904,167.366,53.636,159.946
C01653=1016.283,176.478,374.924,167.361,53.646,159.947
C01654=1016.278,176.229,374.945,167.358,53.657,159.949
C01655=1016.273,175.980,374.966,167.353,53.667,159.950
C01656=1016.269,175.731,374.987,167.350,53.677,159.951
C01657=1016.265,175.482,375.008,167.345,53.688,159.952
C01658=1016.259,175.232,375.028,167.341,53.698,159.954
C01659=1016.255,174.983,375.049,167.337,53.708,159.955
C01660=1016.250,174.735,375.070,167.333,53.718,159.956
C01661=1016.245,174.486,375.092,167.330,53.728,159.957
C01662=1016.241,174.236,375.113,167.325,53.739,159.959
C01663=1016.236,173.988,375.133,167.322,53.749,159.960
C01664=1016.232,173.739,375.154,167.317,53.759,159.961
C01665=1016.226,173.489,375.175,167.314,53.769,159.962
C01666=1016.222,173.241,375.195,167.309,53.780,159.964
C01667=1016.218,172.991,375.216,167.306,53.790,159.965
C01668=1016.213,172.742,375.237,167.302,53.800,159.966
C01669=1016.208,172.493,375.258,167.298,53.811,159.967
C01670=1016.204,172.244,375.279,167.294,53.821,159.969
C01671=1016.199,171.995,375.300,167.290,53.831,159.970
C01672=1016.195,171.746,375.320,167.286,53.841,159.971
C01673=1016.190,171.496,375.340,167.283,53.851,159.972
C01674=1016.185,171.216,375.364,167.277,53.863,159.974
C01675=1016.180,170.935,375.388,167.274,53.875,159.975
C01676=1016.175,170.655,375.410,167.269,53.886,159.977
C01677=1016.170,170.375,375.434,167.265,53.898,159.978
C01678=1016.164,170.126,375.455,167.261,53.908,159.979
C01679=1016.161,169.876,375.475,167.257,53.918,159.981
C01680=1016.156,169.627,375.496,167.253,53.928,159.982
C01681=1016.151,169.378,375.517,167.250,53.939,159.983
C01682=1016.147,169.129,375.537,167.245,53.949,159.984
C01683=1016.142,168.880,375.558,167.242,53.959,159.986
C01684=1016.138,168.631,375.579,167.238,53.969,159.987
C01685=1016.133,168.382,375.600,167.234,53.980,159.988
C01686=1016.128,168.132,375.620,167.230,53.990,159.989
C01687=1016.125,167.883,375.641,167.227,54.000,159.991
C01688=1016.119,167.634,375.661,167.222,54.011,159.992
C01689=1016.115,167.385,375.682,167.219,54.021,159.993
C01690=1016.111,167.136,375.703,167.216,54.031,159.995
C01691=1016.106,166.888,375.723,167.211,54.042,159.996
C01692=1016.102,166.638,375.744,167.208,54.052,159.997
C01693=1016.097,166.389,375.764,167.204,54.062,159.998
C01694=1016.093,166.140,375.785,167.201,54.072,160.000
C01695=1016.089,165.891,375.806,167.196,54.083,160.001
C01696=1016.084,165.641,375.826,167.192,54.092,160.002
C01697=1016.080,165.392,375.846,167.189,54.102,160.003
C01698=1016.075,165.143,375.867,167.185,54.112,160.005
C01699=1016.071,164.895,375.888,167.181,54.123,160.006
C01700=1016.066,164.645,375.908,167.178,54.133,160.007
C01701=1016.062,164.396,375.928,167.174,54.143,160.008
C01702=1016.058,164.147,375.950,167.171,54.153,160.010
C01703=1016.053,163.898,375.970,167.166,54.164,160.011
C01704=1016.049,163.648,375.990,167.163,54.174,160.012
C01705=1016.044,163.400,376.010,167.159,54.184,160.013
C01706=1016.039,163.150,376.031,167.156,54.194,160.015
C01707=1016.036,162.901,376.052,167.152,54.205,160.016
C01708=1016.031,162.652,376.072,167.148,54.215,160.017
C01709=1016.027,162.403,376.093,167.145,54.225,160.019
C01710=1016.022,162.153,376.113,167.141,54.235,160.020
C01711=1016.018,161.905,376.133,167.137,54.245,160.021
C01712=1016.013,161.656,376.154,167.133,54.256,160.022
C01713=1016.009,161.406,376.174,167.130,54.266,160.023
C01714=1016.005,161.157,376.195,167.126,54.276,160.025
C01715=1016.000,160.908,376.215,167.123,54.286,160.026
C01716=1015.996,160.659,376.236,167.119,54.296,160.027
C01717=1015.992,160.411,376.256,167.116,54.307,160.029
C01718=1015.987,160.161,376.276,167.112,54.317,160.030
C01719=1015.983,159.912,376.296,167.108,54.327,160.031
C01720=1015.978,159.662,376.317,167.104,54.337,160.032
C01721=1015.975,159.413,376.338,167.101,54.347,160.034
C01722=1015.970,159.164,376.357,167.098,54.357,160.035
C01723=1015.966,158.915,376.378,167.094,54.368,160.036
C01724=1015.961,158.666,376.398,167.091,54.378,160.038
C01725=1015.957,158.417,376.418,167.088,54.388,160.039
C01726=1015.952,158.167,376.438,167.083,54.399,160.040
C01727=1015.948,157.919,376.458,167.080,54.409,160.041
C01728=1015.943,157.669,376.478,167.076,54.419,160.043
C01729=1015.938,157.420,376.498,167.072,54.430,160.044
C01730=1015.934,157.172,376.518,167.069,54.440,160.045
C01731=1015.930,156.922,376.538,167.066,54.451,160.047
C01732=1015.925,156.673,376.558,167.062,54.461,160.048
C01733=1015.921,156.424,376.577,167.058,54.472,160.049
C01734=1015.916,156.174,376.598,167.055,54.482,160.051
C01735=1015.911,155.925,376.617,167.051,54.492,160.052
C01736=1015.907,155.676,376.637,167.048,54.502,160.053
C01737=1015.902,155.427,376.657,167.044,54.513,160.054
C01738=1015.897,155.146,376.679,167.040,54.525,160.056
C01739=1015.892,154.865,376.701,167.036,54.536,160.058
C01740=1015.887,154.584,376.724,167.032,54.548,160.059
C01741=1015.882,154.304,376.746,167.028,54.560,160.061
C01742=1015.878,154.055,376.766,167.025,54.570,160.062
C01743=1015.873,153.806,376.785,167.022,54.581,160.063
C01744=1015.868,153.556,376.805,167.018,54.591,160.065
C01745=1015.864,153.307,376.825,167.014,54.602,160.066
C01746=1015.859,153.059,376.845,167.011,54.612,160.067
C01747=1015.854,152.809,376.865,167.007,54.622,160.068
C01748=1015.850,152.560,376.884,167.004,54.632,160.070
C01749=1015.846,152.311,376.904,167.001,54.643,160.071
C01750=1015.841,152.062,376.923,166.996,54.653,160.072
C01751=1015.836,151.812,376.943,166.994,54.664,160.074
C01752=1015.832,151.563,376.962,166.990,54.675,160.075
C01753=1015.828,151.314,376.982,166.987,54.685,160.076
C01754=1015.823,151.065,377.001,166.983,54.696,160.078
C01755=1015.818,150.815,377.021,166.979,54.706,160.079
C01756=1015.814,150.566,377.041,166.976,54.716,160.080
C01757=1015.810,150.317,377.060,166.973,54.726,160.082
C01758=1015.805,150.068,377.080,166.969,54.737,160.083
C01759=1015.800,149.818,377.099,166.965,54.747,160.084
C01760=1015.796,149.569,377.119,166.962,54.758,160.086
C01761=1015.792,149.320,377.138,166.959,54.769,160.087
C01762=1015.787,149.071,377.158,166.956,54.779,160.088
C01763=1015.783,148.822,377.177,166.953,54.789,160.090
C01764=1015.778,148.572,377.197,166.948,54.800,160.091
C01765=1015.773,148.324,377.216,166.945,54.810,160.092
C01766=1015.769,148.075,377.236,166.942,54.820,160.094
C01767=1015.765,147.825,377.254,166.938,54.831,160.095
C01768=1015.760,147.576,377.274,166.935,54.841,160.096
C01769=1015.755,147.326,377.294,166.932,54.851,160.098
C01770=1015.751,147.077,377.313,166.928,54.863,160.099
C01771=1015.747,146.828,377.333,166.925,54.873,160.100
C01772=1015.742,146.579,377.352,166.922,54.883,160.102
C01773=1015.738,146.330,377.371,166.918,54.894,160.103
C01774=1015.733,146.081,377.390,166.915,54.904,160.104
C01775=1015.728,145.831,377.409,166.912,54.914,160.106
C01776=1015.724,145.582,377.429,166.909,54.925,160.107
C01777=1015.719,145.333,377.448,166.904,54.935,160.108
C01778=1015.715,145.084,377.468,166.901,54.946,160.110
C01779=1015.710,144.834,377.486,166.899,54.957,160.111
C01780=1015.706,144.585,377.506,166.895,54.967,160.113
C01781=1015.702,144.336,377.525,166.892,54.977,160.114
C01782=1015.696,144.086,377.544,166.888,54.988,160.115
C01783=1015.692,143.837,377.563,166.885,54.998,160.116
C01784=1015.687,143.588,377.582,166.881,55.009,160.118
C01785=1015.683,143.339,377.601,166.879,55.020,160.119
C01786=1015.678,143.090,377.620,166.875,55.030,160.121
C01787=1015.674,142.841,377.640,166.871,55.041,160.122
C01788=1015.669,142.591,377.658,166.868,55.051,160.123
C01789=1015.665,142.342,377.677,166.865,55.061,160.125
C01790=1015.661,142.093,377.697,166.862,55.072,160.126
C01791=1015.655,141.843,377.715,166.858,55.082,160.127
C01792=1015.651,141.594,377.735,166.856,55.093,160.129
C01793=1015.647,141.345,377.753,166.853,55.104,160.130
C01794=1015.642,141.096,377.772,166.848,55.114,160.131
C01795=1015.637,140.847,377.792,166.845,55.125,160.133
C01796=1015.633,140.597,377.811,166.842,55.135,160.134
C01797=1015.628,140.348,377.829,166.839,55.145,160.136
C01798=1015.624,140.099,377.848,166.836,55.156,160.137
C01799=1015.619,139.850,377.867,166.832,55.166,160.138
C01800=1015.615,139.601,377.887,166.829,55.176,160.140
C01801=1015.611,139.351,377.905,166.827,55.188,160.141
C01802=1015.606,139.106,377.924,166.823,55.197,160.142
C01803=1015.602,138.863,377.943,166.820,55.208,160.144
C01804=1015.598,138.618,377.961,166.817,55.218,160.145
C01805=1015.594,138.374,377.979,166.813,55.228,160.146
C01806=1015.588,138.130,377.998,166.810,55.239,160.148
C01807=1015.584,137.886,378.016,166.807,55.249,160.149
C01808=1015.580,137.641,378.035,166.804,55.259,160.150
C01809=1015.575,137.397,378.054,166.801,55.270,160.152
